// TIA Portal V19 export
FUNCTION_BLOCK "A0302_PareggiatoreCoda_FB"   // FB118, LAD
// stored: MemoryReserve 100, SetENOAutomatically false
   VAR_INPUT
      AreaInterface : "AreaInterface";
      ZSI : "udt_ZoneSafetyInterface";
      DSI_Feed : "udt_DeviceSafetyInterface";
      DSI_Valve : "udt_DeviceSafetyInterface";
      DSI_OilValve : "udt_DeviceSafetyInterface";
      Drive : "TAx_DriveInterface";
      DataIn : Struct
         OP_MoveToPos : Bool;
         BattutaVrt : Struct
            OP : "OP_PB";
         END_STRUCT;
         PareggLong : Struct
            OP : "OP_PB";
            AnalSens : Int;
         END_STRUCT;
         Sens { ExternalWritable := 'False'} : Struct
            FTC_Ingombro_In : Bool;   // 2012BF1 - I50.0
            FTC_Ingombro_Out : Bool;   // 2012BF2 - I50.1
            PresenzaMat : Bool;   // FC presenza materiale agganciato lato paregg coda
            FC_Aticoll_Spalla : Bool;
         END_STRUCT;
      END_STRUCT;
      CIn : Struct
         Manager : Struct
            EnableStopDoorOpeningReq { ExternalAccessible := 'False'; ExternalVisible := 'False'; ExternalWritable := 'False'} : Bool;
            EnableStopInPhase { ExternalAccessible := 'False'; ExternalVisible := 'False'; ExternalWritable := 'False'} : Bool;
            EnableStopProgrammed { ExternalAccessible := 'False'; ExternalVisible := 'False'; ExternalWritable := 'False'} : Bool;
            Control_ON { ExternalAccessible := 'False'; ExternalVisible := 'False'; ExternalWritable := 'False'} : Bool;
            MoveToPos { ExternalAccessible := 'False'; ExternalVisible := 'False'; ExternalWritable := 'False'} : Bool;
            Pos { ExternalAccessible := 'False'; ExternalVisible := 'False'; ExternalWritable := 'False'} : LReal;
            Speed : LReal;
            Bloccaggio { ExternalAccessible := 'False'; ExternalVisible := 'False'; ExternalWritable := 'False'} : Struct
               Rest : Bool;
               Work : Bool;
            END_STRUCT;
            BattutaVrt { ExternalAccessible := 'False'; ExternalVisible := 'False'; ExternalWritable := 'False'} : Struct
               Rest : Bool;
               Work : Bool;
            END_STRUCT;
            PareggLong { ExternalAccessible := 'False'; ExternalVisible := 'False'; ExternalWritable := 'False'} : Struct
               Rest : Bool;
               Work : Bool;
            END_STRUCT;
         END_STRUCT;
         SemiAut_Pb { ExternalWritable := 'False'} : Bool;
         Bordatrice : Struct
            Ax : "Positioning_EPOS_Machine_COut";
            Sts : Struct
               PosTargetEnable : Bool;
               PosTarget_Reached : Bool;
               In_W_Pos : Bool;
               AtRest : Bool;
            END_STRUCT;
            RegSpalla : Struct
               Infeed_ReqON : Bool;
            END_STRUCT;
         END_STRUCT;
         Rulliera { ExternalWritable := 'False'} : Struct
            Ax_1 : "SpeedMachine_COut";
            Ax_2 : "SpeedMachine_COut";
            Centratori : "ValveMachine_COut";
            Coda : Struct
               Sens : Struct
                  FTC_Rall : Bool;   // Sensori presenza materiale banco rallentamento ingresso
                  FTC_Prox_Ing : Bool;   // Sensori presenza materiale banco limite ingresso
               END_STRUCT;
            END_STRUCT;
            Centro : Struct
               Sens : Struct
                  FTC_Centrale : Bool;   // 2010BF1 - I50.2
               END_STRUCT;
            END_STRUCT;
         END_STRUCT;
         CarroPareggCoda : Struct
            Pareggia : Bool;   // Bit di abilitazione pareggiamento - prende la misura del beam e controlla la tolleranza
            OilInTargetPressure { ExternalWritable := 'False'} : Bool;
         END_STRUCT;
         CarroPareggTesta { ExternalWritable := 'False'} : Struct
            Sens : Struct
               FTC1_Rall : Bool;   // 2010BF2 - I50.3
               FTC2_Prox_Ls : Bool;   // 2010BF3 - I50.4
               PresenzaMat : Bool;   // FC presenza materiale agganciato lato paregg testa
            END_STRUCT;
         END_STRUCT;
         CarriPareggiatori : Struct
            ZoneA0302Entry_Empty { ExternalWritable := 'False'} : Bool;
            ZoneA0302Exit_Empty { ExternalWritable := 'False'} : Bool;
            RequestNewPosition : Bool;
         END_STRUCT;
         Spalle : Struct
            Coda : Struct
               ActualPos : LReal;
            END_STRUCT;
            Testa : Struct
               ActualPos : LReal;
            END_STRUCT;
         END_STRUCT;
         Manipolatore : Struct
            Sollevatore : "ValveMachine_COut";
         END_STRUCT;
         Centratori : Struct
            Sollevamento : "ValveMachine_COut";
         END_STRUCT;
      END_STRUCT;
      Config : Struct
         Ax : "Positioning_DOL_Machine_Config";
         Bloccaggio : "ValveMachine_Config";
         BattutaVerticale : "ValveMachine_Config";
         PareggiatoreLong : "ValveMachine_Config";
         PosPareggiatore : Struct
            QuotaMin_Work : LReal;
            QuotaMax_Work : LReal;
         END_STRUCT;
         MinDistanzaConSpalla : LReal;
         DelayMissingCondition : Time;
      END_STRUCT;
      HWID : Struct
         Ax_TEL1 : HW_SUBMODULE;
         Enc_IO : HW_SUBMODULE;
      END_STRUCT;
   END_VAR
   VAR_OUTPUT
      MachineInterface : "MachineInterface";
      COut : Struct
         Ax : "Positioning_DOL_Machine_COut";
         Bloccaggio : "ValveMachine_COut";
         BattutaVerticale : "ValveMachine_COut";
         PareggiatoreLong : "ValveMachine_COut";
         Ax_InWPos : Bool;
         Anticipi : Struct
            Work : Struct
               BattutaVrt : Bool;
               PareggLong : Bool;
            END_STRUCT;
            Rest : Struct
               BattutaVrt : Bool;
               PareggLong : Bool;
            END_STRUCT;
         END_STRUCT;
      END_STRUCT;
   END_VAR
   VAR_IN_OUT
      Par : Struct
         Ax : "Positioning_DOL_Machine_Par";
         Ax_Pers : "Positioning_DOL_Machine_Pers_Data";
         Enc : "PosFbk_RTN";
         Ax_Aut : "A0301_Mach_Speed_Par";
         Bloccaggio_Sens : Struct
            "2191B1" : "Analogic_SensorManagement_Par";
            SogliaWork : Real;
         END_STRUCT;
         CarroPareggCoda : Struct
            Delay_StartMove : Time;
            Preset : LReal;
         END_STRUCT;
         Cremaliera : Struct
            Modulo : LReal;
            Passo : LReal;
         END_STRUCT;
      END_STRUCT;
      Par_Sens : Struct
         AI : "Analogic_SensorManagement_Par";
      END_STRUCT;
      Data_Sens : "Analogic_SensorManagement_Data";
      Par_MachSens : "A0301_Mach_Sens_Par";
      IEC_SP : Struct
         FTC_Input : Struct
            TON_PT : Time;
            TOF_PT : Time;
         END_STRUCT;
         FTC_Output : Struct
            TON_PT : Time;
            TOF_PT : Time;
         END_STRUCT;
         FTC_PresentMat : Struct
            TON_PT : Time;
            TOF_PT : Time;
         END_STRUCT;
         Check_2119B1 : Struct
            TON_PT : Time;
         END_STRUCT;
      END_STRUCT;
   END_VAR
   VAR
      Alarm : Struct
         Ax : "Positioning_DOL_Machine_Alr";
         Enc : "PosFbk_Encoder_Alr";
         Bloccaggio : "ValveAlr";
         BattutaVerticale : "ValveAlr";
         PareggiatoreLong : "ValveAlr";
         PareggLong_AnalSens_Issue : Bool;
         SensFC_Aticoll_Spalla : Bool;
         Bloccaggio_AnalSens_Issue : Bool;   // Errore soglia lettura pressione su bloccaggio cremaliera
      END_STRUCT;
      Warning : Struct
         Ax : "Positioning_DOL_Machine_Wng";
         Bloccaggio : "ValveMachine_Wng";
         BattutaVerticale : "ValveMachine_Wng";
         PareggiatoreLongitudinale : "ValveMachine_Wng";
         PosPareggiatoreLong : "Analogic_SensorManagement_Warning";
         MissingCnd : Struct
            OP_REST_BattutaVrt : Bool;   // Mancanza comando arresto
            OP_WORK_BattutaVrt : Bool;   // Mancanza consenso lavoro
            OP_REST_PareggLong : Bool;   // Mancanza comando arresto
            OP_WORK_PareggLong : Bool;   // Mancanza consenso lavoro
            OP_REST_Bloccaggio : Bool;   // Mancanza comando arresto
            OP_WORK_Bloccaggio : Bool;   // Mancanza consenso lavoro
         END_STRUCT;
         SW_Limit_AntiCollision : Bool;
      END_STRUCT;
      HMI : Struct
         AnalogSensor : "AnalogSens_HmiData";
         Ax : Struct
            PbPreset : Bool;
            B_Preset_UM2 : Bool;
            PresetValue : LReal;
         END_STRUCT;
      END_STRUCT;
      Sts : Struct
         ReadyForMove : Bool;   // Pronto al movimento
         OP_PCoda_CanMoveFreely : Bool;
         OP_Ax_CanMoveFreely : Bool;
         Op_MoveToPos_Cnd : Bool;
         BattutaVrt : Struct
            OP_Rest_Cnd : Bool;
            Op_Work_Cnd : Bool;
         END_STRUCT;
         PareggLong : Struct
            OP_Rest_Cnd : Bool;
            Op_Work_Cnd : Bool;
         END_STRUCT;
      END_STRUCT;
      Ctrl : Struct
         BattutaVrt : Struct
            OP_Rest_Man : Bool;
            OP_Work_Man : Bool;
            OP_Rest_Aut : Bool;
            OP_Work_Aut : Bool;
            OP_Rest : Bool;
            OP_Work : Bool;
         END_STRUCT;
         PareggLong : Struct
            CheckMesure : Bool;   // Bit che determina l'uscita del pareggiatore e Controlla misura Blea nel manager
            OP_Rest_Aut : Bool;
            OP_Work_Aut : Bool;
            OP_Rest_Man : Bool;
            OP_Work_Man : Bool;
            OP_Rest : Bool;
            OP_Work : Bool;
         END_STRUCT;
         Ax : Struct
            OP_MoveToPos_Man : Bool;
            OP_MoveToPos_Aut : Bool;
            OP_MoveToPos : Bool;
         END_STRUCT;
      END_STRUCT;
      AUX : Struct
         OP_MoveToPos : Bool;
         BattutaVrt : Struct
            OP_Rest : Bool;
            OP_Work : Bool;
         END_STRUCT;
         PareggLong : Struct
            OP_Rest : Bool;
            OP_Work : Bool;
         END_STRUCT;
      END_STRUCT;
      Ax { S7_SetPoint := 'True'} : "Positioning_DOL_Machine_FB";   // Asse di movimento carro pareggiatore su cremaliera
      Enc : "PosFbk_SickAFM60";
      Enc_ITF : "PosFbk_ITF";
      Bloccaggio { S7_SetPoint := 'True'} : "ValveMachine_FB";   // Bloccaggio cremaliera
      BattutaVerticale { S7_SetPoint := 'True'} : "ValveMachine_FB";   // Battuta verticale
      PareggiatoreLong { S7_SetPoint := 'True'} : "ValveMachine_FB";   // Pareggiatore longitudinale
      PosPareggLong { S7_SetPoint := 'True'} : "Analogic_SensorManagement";   // Sensore di posizione pareggiatore
      TON_PareggLong : Struct
         OP_REST_MissingCnd { S7_SetPoint := 'True'} : TON_TIME;
         OP_WORK_MissingCnd { S7_SetPoint := 'True'} : TON_TIME;
      END_STRUCT;
      TON_BattutaVrt : Struct
         OP_REST_MissingCnd { S7_SetPoint := 'True'} : TON_TIME;
         OP_WORK_MissingCnd { S7_SetPoint := 'True'} : TON_TIME;
      END_STRUCT;
      TON_Bloccaggio : Struct
         OP_REST_MissingCnd { S7_SetPoint := 'True'} : TON_TIME;
         OP_WORK_MissingCnd { S7_SetPoint := 'True'} : TON_TIME;
      END_STRUCT;
      IEC_FTC_Input : Struct
         TON_Delay : IEC_TIMER;
         TOF_Delay { S7_SetPoint := 'True'} : IEC_TIMER;
         FTC_On { S7_SetPoint := 'True'} : Bool;
      END_STRUCT;
      IEC_FTC_Output : Struct
         TON_Delay : IEC_TIMER;
         TOF_Delay { S7_SetPoint := 'True'} : IEC_TIMER;
         FTC_On { S7_SetPoint := 'True'} : Bool;
      END_STRUCT;
      IEC_FTC_PresentMat : Struct
         TON_Delay : IEC_TIMER;
         TOF_Delay { S7_SetPoint := 'True'} : IEC_TIMER;
         FTC_On { S7_SetPoint := 'True'} : Bool;
      END_STRUCT;
      IEC_DelayCheck_2119B1 : IEC_TIMER;
      Bloccaggio_AnalSens { S7_SetPoint := 'True'} : "AnalogThreshold";
      CarroCoda { ExternalAccessible := 'False'; ExternalVisible := 'False'; ExternalWritable := 'False'} : Struct
         RimanenzaPos : LReal;
         PassoReq : LReal;
         PosBattutePz : LReal;
         SemiBeamLen : LReal;
         NrPassiReq : LReal;
         Pos : LReal;   // Posizione calcolata in funzione della cremaliera
      END_STRUCT;
      TON_DistanzaOK : IEC_TIMER;
      TON_Anticipi : Struct
         Rest : Struct
            BattutaVrt { S7_SetPoint := 'True'} : IEC_TIMER;
            PareggLong : IEC_TIMER;
         END_STRUCT;
         Work : Struct
            PareggLong : IEC_TIMER;
            BattutaVrt { S7_SetPoint := 'True'} : IEC_TIMER;
         END_STRUCT;
      END_STRUCT;
   END_VAR
   VAR_TEMP
      PE : Struct
         OP_MoveToPos : Bool;
         BattutaVrt : Struct
            OP_Rest : Bool;
            OP_Work : Bool;
         END_STRUCT;
         PareggLong : Struct
            OP_Rest : Bool;
            OP_Work : Bool;
         END_STRUCT;
      END_STRUCT;
      ActualDifference : LReal;
   END_VAR
   VAR CONSTANT
      RACK_STEP : LReal;   // Passo Cremagliera mm
   END_VAR
   VAR_TEMP   // added for the SCL form of the ladder/FBD networks
      _w1 : Bool;
      _w2 : Bool;
      _w3 : Bool;
      _w4 : Bool;
      _w5 : Bool;
      _w6 : Bool;
      _w7 : Bool;
      _w8 : Bool;
      _w9 : Bool;
      _w10 : Bool;
      _w11 : Bool;
      _w12 : Bool;
   END_VAR
BEGIN

REGION Network 1 (SCL): Reset allarmi
   IF #AreaInterface.RstAlarms THEN
       #Alarm.PareggLong_AnalSens_Issue := FALSE;
       #Alarm.SensFC_Aticoll_Spalla := FALSE;
       #Alarm.Bloccaggio_AnalSens_Issue := FALSE;
   END_IF;
END_REGION

REGION Network 2: <+>
END_REGION

REGION Network 3: Anticipi Movimento LAVORO
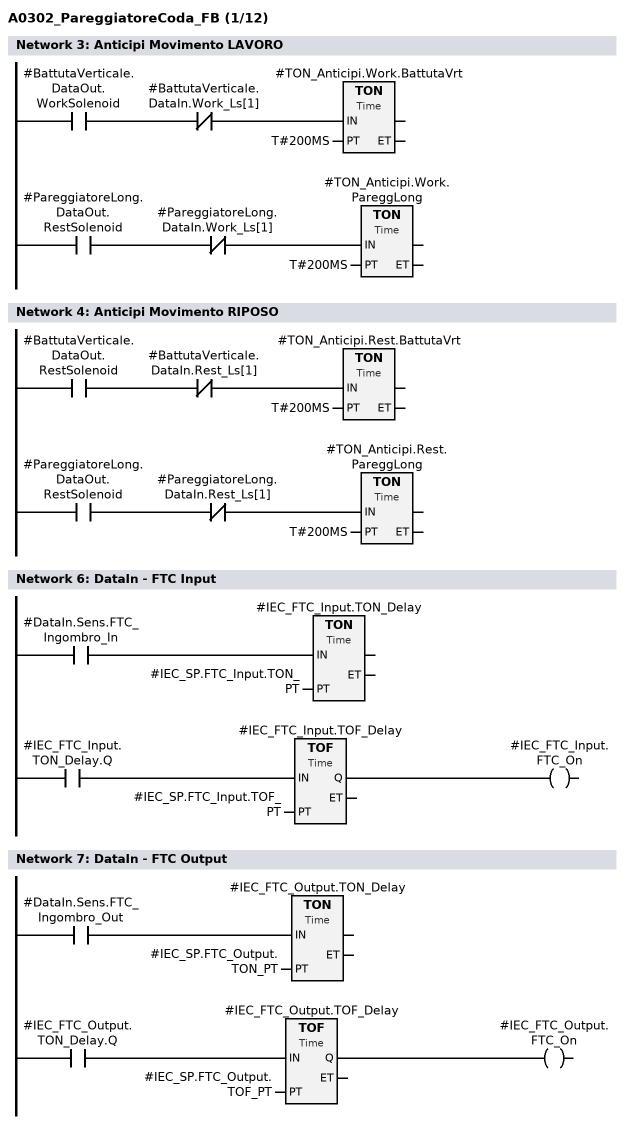
   RUNG wire#powerrail
      Contact( #BattutaVerticale.DataOut.WorkSolenoid )
      I_Contact( #BattutaVerticale.DataIn.Work_Ls[1] )
      { S7_Templates := "time_type := Time" } #TON_Anticipi.Work.BattutaVrt.TON(pt := T#200MS, et =>)
   END_RUNG
   RUNG wire#powerrail
      Contact( #PareggiatoreLong.DataOut.RestSolenoid )
      I_Contact( #PareggiatoreLong.DataIn.Work_Ls[1] )
      { S7_Templates := "time_type := Time" } #TON_Anticipi.Work.PareggLong.TON(pt := T#200MS, et =>)
   END_RUNG
   // the same network as SCL:
   #TON_Anticipi.Work.BattutaVrt.TON(IN := #BattutaVerticale.DataOut.WorkSolenoid AND NOT #BattutaVerticale.DataIn.Work_Ls[1],
                           PT := T#200MS);
   #TON_Anticipi.Work.PareggLong.TON(IN := #PareggiatoreLong.DataOut.RestSolenoid AND NOT #PareggiatoreLong.DataIn.Work_Ls[1],
                           PT := T#200MS);
END_REGION

REGION Network 4: Anticipi Movimento RIPOSO
   RUNG wire#powerrail
      Contact( #BattutaVerticale.DataOut.RestSolenoid )
      I_Contact( #BattutaVerticale.DataIn.Rest_Ls[1] )
      { S7_Templates := "time_type := Time" } #TON_Anticipi.Rest.BattutaVrt.TON(pt := T#200MS, et =>)
   END_RUNG
   RUNG wire#powerrail
      Contact( #PareggiatoreLong.DataOut.RestSolenoid )
      I_Contact( #PareggiatoreLong.DataIn.Rest_Ls[1] )
      { S7_Templates := "time_type := Time" } #TON_Anticipi.Rest.PareggLong.TON(pt := T#200MS, et =>)
   END_RUNG
   // the same network as SCL:
   #TON_Anticipi.Rest.BattutaVrt.TON(IN := #BattutaVerticale.DataOut.RestSolenoid AND NOT #BattutaVerticale.DataIn.Rest_Ls[1],
                           PT := T#200MS);
   #TON_Anticipi.Rest.PareggLong.TON(IN := #PareggiatoreLong.DataOut.RestSolenoid AND NOT #PareggiatoreLong.DataIn.Rest_Ls[1],
                           PT := T#200MS);
END_REGION

REGION Network 5: <+>
END_REGION

REGION Network 6: DataIn - FTC Input
   RUNG wire#powerrail
      Contact( #DataIn.Sens.FTC_Ingombro_In )
      { S7_Templates := "time_type := Time" } #IEC_FTC_Input.TON_Delay.TON(pt := #IEC_SP.FTC_Input.TON_PT, et =>)
   END_RUNG
   RUNG wire#powerrail
      Contact( #IEC_FTC_Input.TON_Delay.Q )
      { S7_Templates := "time_type := Time" } #IEC_FTC_Input.TOF_Delay.TOF(pt := #IEC_SP.FTC_Input.TOF_PT, et =>)
      Coil( #IEC_FTC_Input.FTC_On )
   END_RUNG
   // the same network as SCL:
   #IEC_FTC_Input.TON_Delay.TON(IN := #DataIn.Sens.FTC_Ingombro_In, PT := #IEC_SP.FTC_Input.TON_PT);
   #IEC_FTC_Input.TOF_Delay.TOF(IN := #IEC_FTC_Input.TON_Delay.Q, PT := #IEC_SP.FTC_Input.TOF_PT);
   #IEC_FTC_Input.FTC_On := #IEC_FTC_Input.TOF_Delay.Q;
END_REGION

REGION Network 7: DataIn - FTC Output
   RUNG wire#powerrail
      Contact( #DataIn.Sens.FTC_Ingombro_Out )
      { S7_Templates := "time_type := Time" } #IEC_FTC_Output.TON_Delay.TON(pt := #IEC_SP.FTC_Output.TON_PT, et =>)
   END_RUNG
   RUNG wire#powerrail
      Contact( #IEC_FTC_Output.TON_Delay.Q )
      { S7_Templates := "time_type := Time" } #IEC_FTC_Output.TOF_Delay.TOF(pt := #IEC_SP.FTC_Output.TOF_PT, et =>)
      Coil( #IEC_FTC_Output.FTC_On )
   END_RUNG
   // the same network as SCL:
   #IEC_FTC_Output.TON_Delay.TON(IN := #DataIn.Sens.FTC_Ingombro_Out, PT := #IEC_SP.FTC_Output.TON_PT);
   #IEC_FTC_Output.TOF_Delay.TOF(IN := #IEC_FTC_Output.TON_Delay.Q, PT := #IEC_SP.FTC_Output.TOF_PT);
   #IEC_FTC_Output.FTC_On := #IEC_FTC_Output.TOF_Delay.Q;
END_REGION

REGION Network 8: DataIn - FTC Presenza materiale
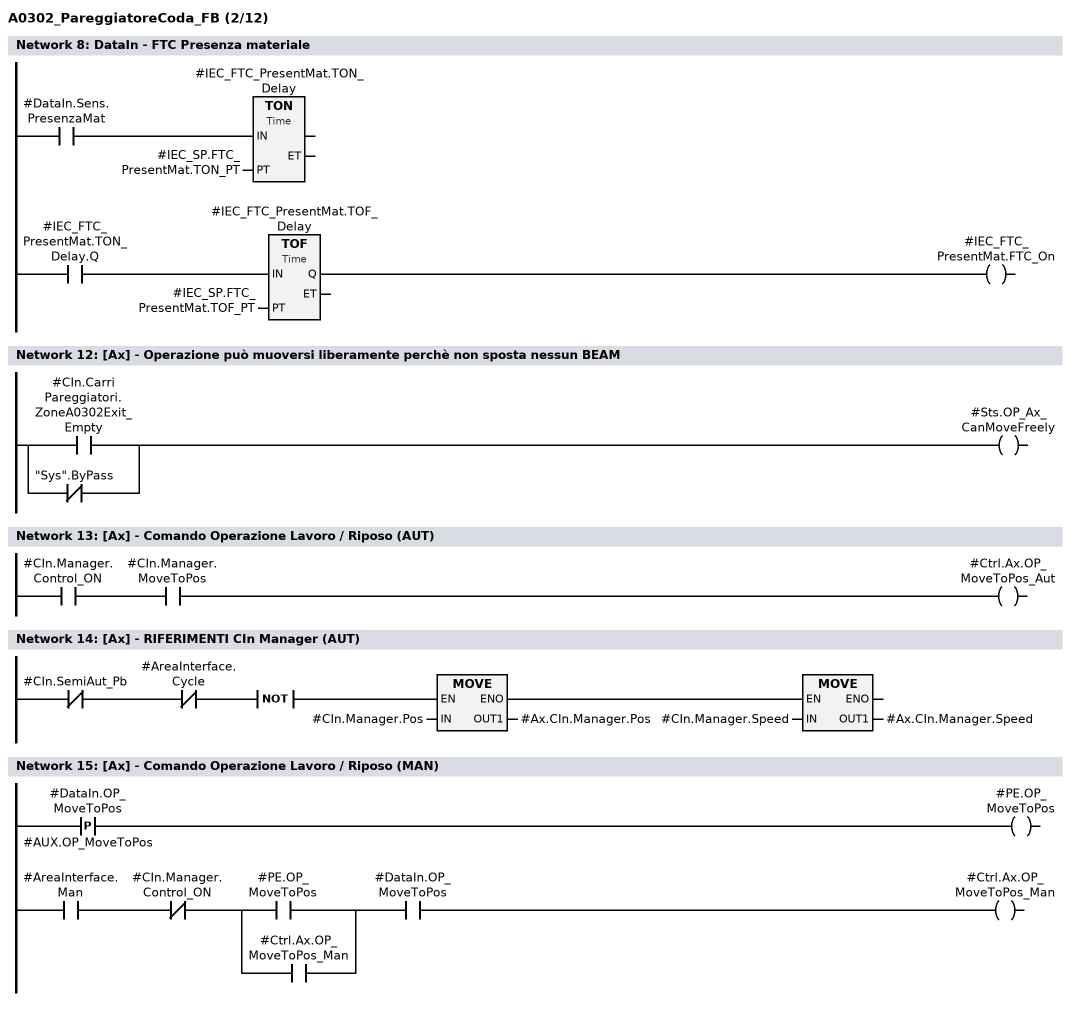
   RUNG wire#powerrail
      Contact( #DataIn.Sens.PresenzaMat )
      { S7_Templates := "time_type := Time" } #IEC_FTC_PresentMat.TON_Delay.TON(pt := #IEC_SP.FTC_PresentMat.TON_PT, et =>)
   END_RUNG
   RUNG wire#powerrail
      Contact( #IEC_FTC_PresentMat.TON_Delay.Q )
      { S7_Templates := "time_type := Time" } #IEC_FTC_PresentMat.TOF_Delay.TOF(pt := #IEC_SP.FTC_PresentMat.TOF_PT, et =>)
      Coil( #IEC_FTC_PresentMat.FTC_On )
   END_RUNG
   // the same network as SCL:
   #IEC_FTC_PresentMat.TON_Delay.TON(IN := #DataIn.Sens.PresenzaMat, PT := #IEC_SP.FTC_PresentMat.TON_PT);
   #IEC_FTC_PresentMat.TOF_Delay.TOF(IN := #IEC_FTC_PresentMat.TON_Delay.Q, PT := #IEC_SP.FTC_PresentMat.TOF_PT);
   #IEC_FTC_PresentMat.FTC_On := #IEC_FTC_PresentMat.TOF_Delay.Q;
END_REGION

REGION Network 9: <+>
END_REGION

REGION Network 10: <<< CARRO PAREGGIATORE CODA >>>
END_REGION

REGION Network 11: <+>
END_REGION

REGION Network 12: [Ax] - Operazione può muoversi liberamente perchè non sposta nessun BEAM
   RUNG wire#powerrail
      Contact( #CIn.CarriPareggiatori.ZoneA0302Exit_Empty )
      wire#w1
      Coil( #Sts.OP_Ax_CanMoveFreely )
   END_RUNG
   RUNG wire#powerrail
      I_Contact( "Sys".ByPass )
   END_RUNG wire#w1
   // the same network as SCL:
   #Sts.OP_Ax_CanMoveFreely := #CIn.CarriPareggiatori.ZoneA0302Exit_Empty OR NOT "Sys".ByPass;
END_REGION

REGION Network 13: [Ax] - Comando Operazione Lavoro / Riposo (AUT)
   RUNG wire#powerrail
      Contact( #CIn.Manager.Control_ON )
      Contact( #CIn.Manager.MoveToPos )
      Coil( #Ctrl.Ax.OP_MoveToPos_Aut )
   END_RUNG
   // the same network as SCL:
   #Ctrl.Ax.OP_MoveToPos_Aut := #CIn.Manager.Control_ON AND #CIn.Manager.MoveToPos;
END_REGION

REGION Network 14: [Ax] - RIFERIMENTI CIn Manager (AUT)
   RUNG wire#powerrail
      I_Contact( #CIn.SemiAut_Pb )
      I_Contact( #AreaInterface.Cycle )
      Not()
      Move(in := #CIn.Manager.Pos, out1 => #Ax.CIn.Manager.Pos)
      Move(in := #CIn.Manager.Speed, out1 => #Ax.CIn.Manager.Speed)
   END_RUNG
   // the same network as SCL:
   IF NOT (NOT #CIn.SemiAut_Pb AND NOT #AreaInterface.Cycle) THEN
       #Ax.CIn.Manager.Pos := #CIn.Manager.Pos;
       #Ax.CIn.Manager.Speed := #CIn.Manager.Speed;
   END_IF;
END_REGION

REGION Network 15: [Ax] - Comando Operazione Lavoro / Riposo (MAN)
   RUNG wire#powerrail
      P_Contact(operand := #DataIn.OP_MoveToPos, bit := #AUX.OP_MoveToPos)
      Coil( #PE.OP_MoveToPos )
   END_RUNG
   RUNG wire#powerrail
      Contact( #AreaInterface.Man )
      I_Contact( #CIn.Manager.Control_ON )
      wire#w1
      Contact( #PE.OP_MoveToPos )
      wire#w2
      Contact( #DataIn.OP_MoveToPos )
      Coil( #Ctrl.Ax.OP_MoveToPos_Man )
   END_RUNG
   RUNG wire#w1
      Contact( #Ctrl.Ax.OP_MoveToPos_Man )
   END_RUNG wire#w2
   // the same network as SCL:
   #_w1 := #DataIn.OP_MoveToPos AND NOT #AUX.OP_MoveToPos;   // rising edge of #DataIn.OP_MoveToPos
   #AUX.OP_MoveToPos := #DataIn.OP_MoveToPos;
   #PE.OP_MoveToPos := #_w1;
   #Ctrl.Ax.OP_MoveToPos_Man := #AreaInterface.Man AND NOT #CIn.Manager.Control_ON AND (#PE.OP_MoveToPos OR #Ctrl.Ax.OP_MoveToPos_Man) AND #DataIn.OP_MoveToPos;
END_REGION

REGION Network 16: <+>
END_REGION

REGION Network 17: [Battuta Vrt + Paregg. Long] - Operazione può muoversi liberamente perchè non sposta nessun BEAM
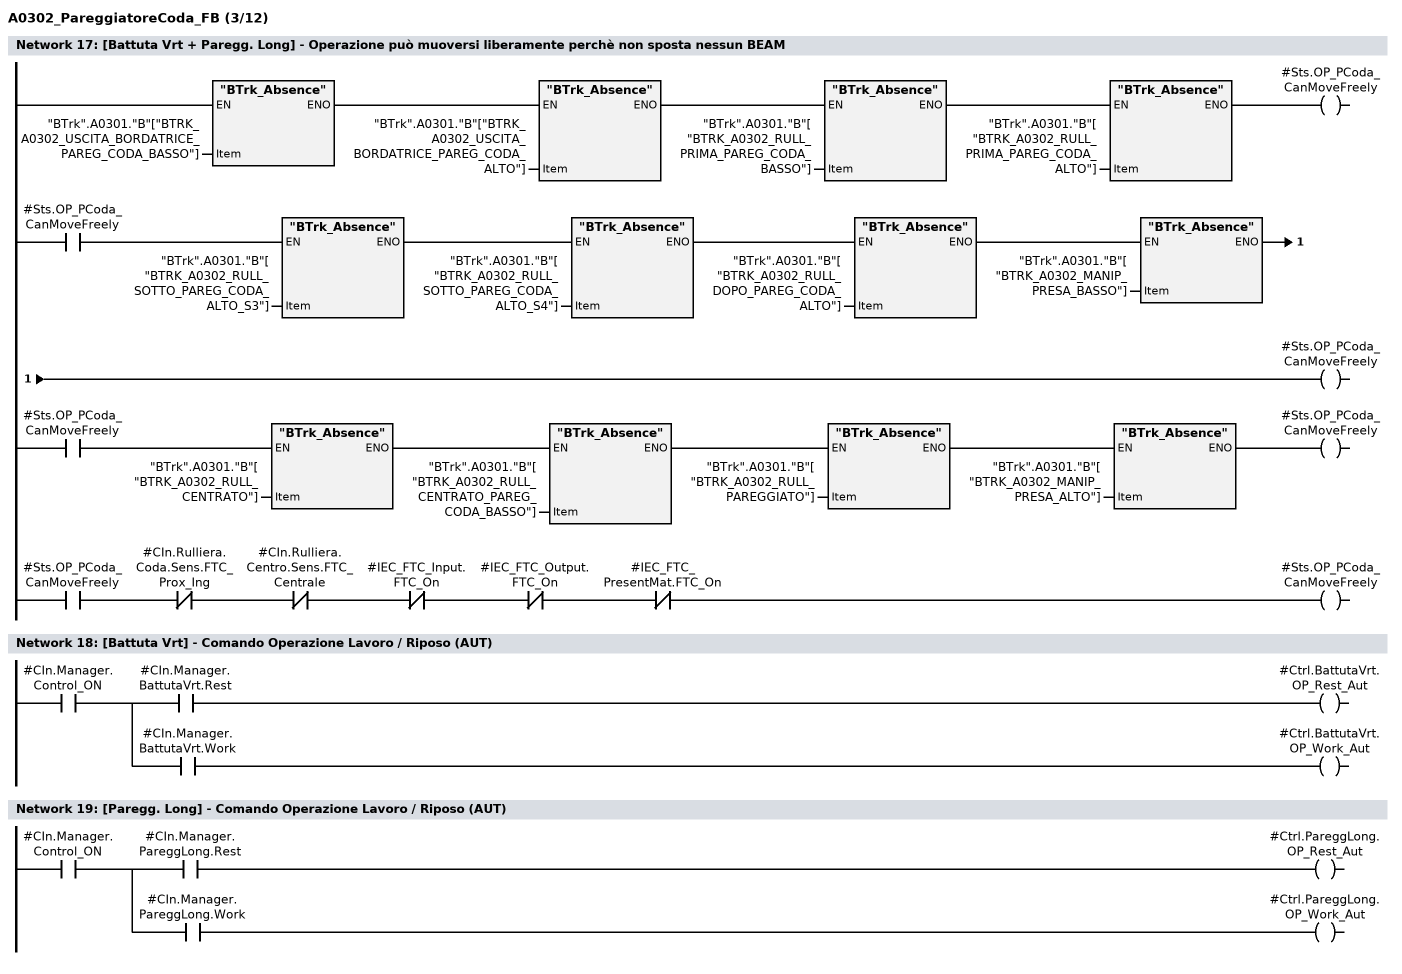
   RUNG wire#powerrail
      "BTrk_Absence"(Item := "BTrk".A0301."B"["BTRK_A0302_USCITA_BORDATRICE_PAREG_CODA_BASSO"])
      "BTrk_Absence"(Item := "BTrk".A0301."B"["BTRK_A0302_USCITA_BORDATRICE_PAREG_CODA_ALTO"])
      "BTrk_Absence"(Item := "BTrk".A0301."B"["BTRK_A0302_RULL_PRIMA_PAREG_CODA_BASSO"])
      "BTrk_Absence"(Item := "BTrk".A0301."B"["BTRK_A0302_RULL_PRIMA_PAREG_CODA_ALTO"])
      Coil( #Sts.OP_PCoda_CanMoveFreely )
   END_RUNG
   RUNG wire#powerrail
      Contact( #Sts.OP_PCoda_CanMoveFreely )
      "BTrk_Absence"(Item := "BTrk".A0301."B"["BTRK_A0302_RULL_SOTTO_PAREG_CODA_ALTO_S3"])
      "BTrk_Absence"(Item := "BTrk".A0301."B"["BTRK_A0302_RULL_SOTTO_PAREG_CODA_ALTO_S4"])
      "BTrk_Absence"(Item := "BTrk".A0301."B"["BTRK_A0302_RULL_DOPO_PAREG_CODA_ALTO"])
      "BTrk_Absence"(Item := "BTrk".A0301."B"["BTRK_A0302_MANIP_PRESA_BASSO"])
      Coil( #Sts.OP_PCoda_CanMoveFreely )
   END_RUNG
   RUNG wire#powerrail
      Contact( #Sts.OP_PCoda_CanMoveFreely )
      "BTrk_Absence"(Item := "BTrk".A0301."B"["BTRK_A0302_RULL_CENTRATO"])
      "BTrk_Absence"(Item := "BTrk".A0301."B"["BTRK_A0302_RULL_CENTRATO_PAREG_CODA_BASSO"])
      "BTrk_Absence"(Item := "BTrk".A0301."B"["BTRK_A0302_RULL_PAREGGIATO"])
      "BTrk_Absence"(Item := "BTrk".A0301."B"["BTRK_A0302_MANIP_PRESA_ALTO"])
      Coil( #Sts.OP_PCoda_CanMoveFreely )
   END_RUNG
   RUNG wire#powerrail
      Contact( #Sts.OP_PCoda_CanMoveFreely )
      I_Contact( #CIn.Rulliera.Coda.Sens.FTC_Prox_Ing )
      I_Contact( #CIn.Rulliera.Centro.Sens.FTC_Centrale )
      I_Contact( #IEC_FTC_Input.FTC_On )
      I_Contact( #IEC_FTC_Output.FTC_On )
      I_Contact( #IEC_FTC_PresentMat.FTC_On )
      Coil( #Sts.OP_PCoda_CanMoveFreely )
   END_RUNG
   // the same network as SCL:
   "BTrk_Absence"(Item := "BTrk".A0301."B"["BTRK_A0302_USCITA_BORDATRICE_PAREG_CODA_BASSO"], ENO => #_w1);
   "BTrk_Absence"(EN := #_w1,
                  Item := "BTrk".A0301."B"["BTRK_A0302_USCITA_BORDATRICE_PAREG_CODA_ALTO"],
                  ENO => #_w2);
   "BTrk_Absence"(EN := #_w2, Item := "BTrk".A0301."B"["BTRK_A0302_RULL_PRIMA_PAREG_CODA_BASSO"], ENO => #_w3);
   "BTrk_Absence"(EN := #_w3, Item := "BTrk".A0301."B"["BTRK_A0302_RULL_PRIMA_PAREG_CODA_ALTO"], ENO => #_w4);
   #Sts.OP_PCoda_CanMoveFreely := #_w4;
   "BTrk_Absence"(EN := #Sts.OP_PCoda_CanMoveFreely,
                  Item := "BTrk".A0301."B"["BTRK_A0302_RULL_SOTTO_PAREG_CODA_ALTO_S3"],
                  ENO => #_w5);
   "BTrk_Absence"(EN := #_w5, Item := "BTrk".A0301."B"["BTRK_A0302_RULL_SOTTO_PAREG_CODA_ALTO_S4"], ENO => #_w6);
   "BTrk_Absence"(EN := #_w6, Item := "BTrk".A0301."B"["BTRK_A0302_RULL_DOPO_PAREG_CODA_ALTO"], ENO => #_w7);
   "BTrk_Absence"(EN := #_w7, Item := "BTrk".A0301."B"["BTRK_A0302_MANIP_PRESA_BASSO"], ENO => #_w8);
   #Sts.OP_PCoda_CanMoveFreely := #_w8;
   "BTrk_Absence"(EN := #Sts.OP_PCoda_CanMoveFreely,
                  Item := "BTrk".A0301."B"["BTRK_A0302_RULL_CENTRATO"],
                  ENO => #_w9);
   "BTrk_Absence"(EN := #_w9,
                  Item := "BTrk".A0301."B"["BTRK_A0302_RULL_CENTRATO_PAREG_CODA_BASSO"],
                  ENO => #_w10);
   "BTrk_Absence"(EN := #_w10, Item := "BTrk".A0301."B"["BTRK_A0302_RULL_PAREGGIATO"], ENO => #_w11);
   "BTrk_Absence"(EN := #_w11, Item := "BTrk".A0301."B"["BTRK_A0302_MANIP_PRESA_ALTO"], ENO => #_w12);
   #Sts.OP_PCoda_CanMoveFreely := #_w12;
   #Sts.OP_PCoda_CanMoveFreely := #Sts.OP_PCoda_CanMoveFreely AND NOT #CIn.Rulliera.Coda.Sens.FTC_Prox_Ing AND NOT #CIn.Rulliera.Centro.Sens.FTC_Centrale AND NOT #IEC_FTC_Input.FTC_On AND NOT #IEC_FTC_Output.FTC_On AND NOT #IEC_FTC_PresentMat.FTC_On;
END_REGION

REGION Network 18: [Battuta Vrt] - Comando Operazione Lavoro / Riposo (AUT)
   RUNG wire#powerrail
      Contact( #CIn.Manager.Control_ON )
      wire#w1
      Contact( #CIn.Manager.BattutaVrt.Rest )
      Coil( #Ctrl.BattutaVrt.OP_Rest_Aut )
   END_RUNG
   RUNG wire#w1
      Contact( #CIn.Manager.BattutaVrt.Work )
      Coil( #Ctrl.BattutaVrt.OP_Work_Aut )
   END_RUNG
   // the same network as SCL:
   #Ctrl.BattutaVrt.OP_Rest_Aut := #CIn.Manager.Control_ON AND #CIn.Manager.BattutaVrt.Rest;
   #Ctrl.BattutaVrt.OP_Work_Aut := #CIn.Manager.Control_ON AND #CIn.Manager.BattutaVrt.Work;
END_REGION

REGION Network 19: [Paregg. Long] - Comando Operazione Lavoro / Riposo (AUT)
   RUNG wire#powerrail
      Contact( #CIn.Manager.Control_ON )
      wire#w1
      Contact( #CIn.Manager.PareggLong.Rest )
      Coil( #Ctrl.PareggLong.OP_Rest_Aut )
   END_RUNG
   RUNG wire#w1
      Contact( #CIn.Manager.PareggLong.Work )
      Coil( #Ctrl.PareggLong.OP_Work_Aut )
   END_RUNG
   // the same network as SCL:
   #Ctrl.PareggLong.OP_Rest_Aut := #CIn.Manager.Control_ON AND #CIn.Manager.PareggLong.Rest;
   #Ctrl.PareggLong.OP_Work_Aut := #CIn.Manager.Control_ON AND #CIn.Manager.PareggLong.Work;
END_REGION

REGION Network 20: <+>
END_REGION

REGION Network 21: [Battuta Vrt] - Comando Operazione Lavoro / Riposo (MAN)
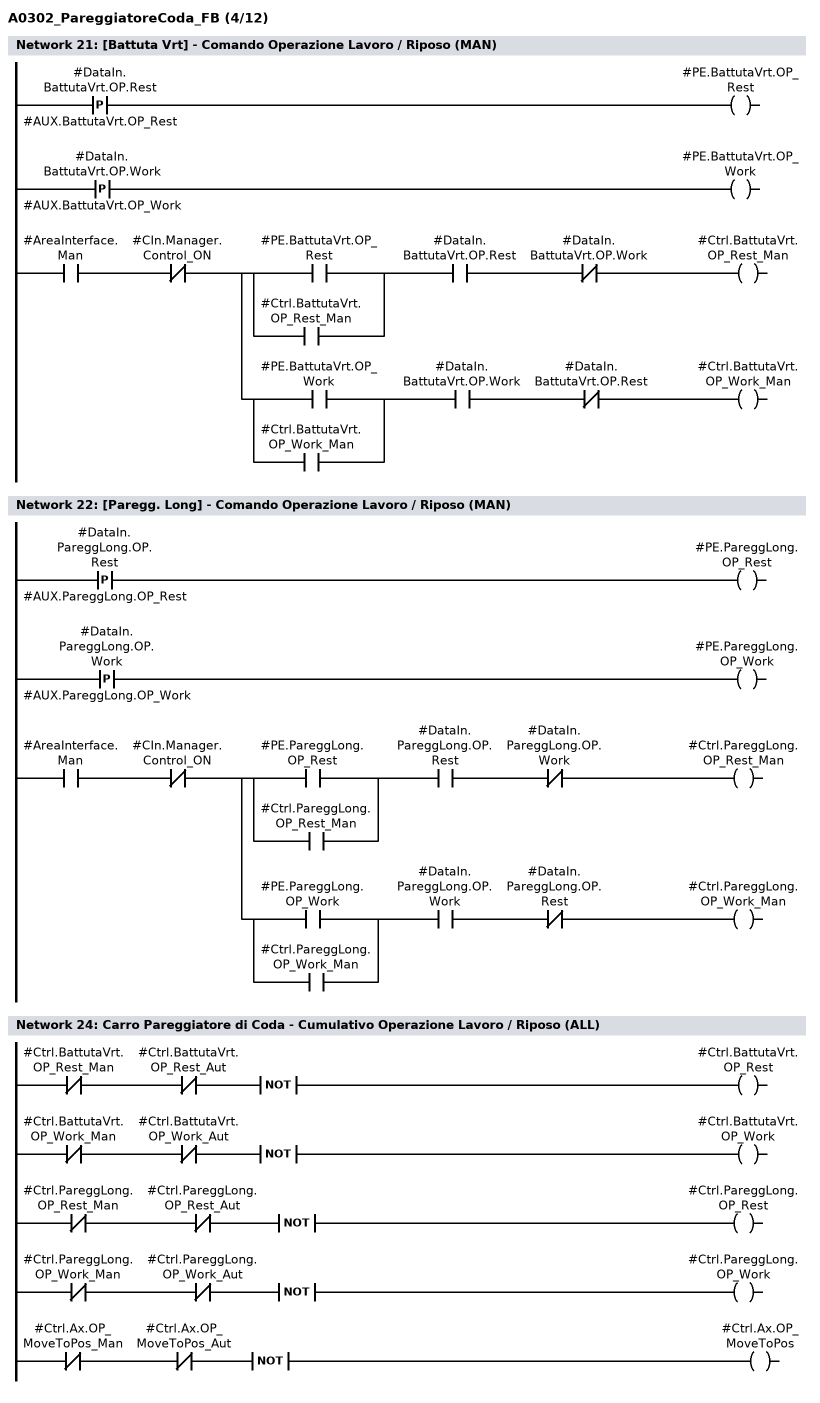
   RUNG wire#powerrail
      P_Contact(operand := #DataIn.BattutaVrt.OP.Rest, bit := #AUX.BattutaVrt.OP_Rest)
      Coil( #PE.BattutaVrt.OP_Rest )
   END_RUNG
   RUNG wire#powerrail
      P_Contact(operand := #DataIn.BattutaVrt.OP.Work, bit := #AUX.BattutaVrt.OP_Work)
      Coil( #PE.BattutaVrt.OP_Work )
   END_RUNG
   RUNG wire#powerrail
      Contact( #AreaInterface.Man )
      I_Contact( #CIn.Manager.Control_ON )
      wire#w1
      Contact( #PE.BattutaVrt.OP_Rest )
      wire#w2
      Contact( #DataIn.BattutaVrt.OP.Rest )
      I_Contact( #DataIn.BattutaVrt.OP.Work )
      Coil( #Ctrl.BattutaVrt.OP_Rest_Man )
   END_RUNG
   RUNG wire#w1
      Contact( #Ctrl.BattutaVrt.OP_Rest_Man )
   END_RUNG wire#w2
   RUNG wire#w1
      Contact( #PE.BattutaVrt.OP_Work )
      wire#w3
      Contact( #DataIn.BattutaVrt.OP.Work )
      I_Contact( #DataIn.BattutaVrt.OP.Rest )
      Coil( #Ctrl.BattutaVrt.OP_Work_Man )
   END_RUNG
   RUNG wire#w1
      Contact( #Ctrl.BattutaVrt.OP_Work_Man )
   END_RUNG wire#w3
   // the same network as SCL:
   #_w1 := #DataIn.BattutaVrt.OP.Rest AND NOT #AUX.BattutaVrt.OP_Rest;   // rising edge of #DataIn.BattutaVrt.OP.Rest
   #AUX.BattutaVrt.OP_Rest := #DataIn.BattutaVrt.OP.Rest;
   #PE.BattutaVrt.OP_Rest := #_w1;
   #_w2 := #DataIn.BattutaVrt.OP.Work AND NOT #AUX.BattutaVrt.OP_Work;   // rising edge of #DataIn.BattutaVrt.OP.Work
   #AUX.BattutaVrt.OP_Work := #DataIn.BattutaVrt.OP.Work;
   #PE.BattutaVrt.OP_Work := #_w2;
   #_w3 := #AreaInterface.Man AND NOT #CIn.Manager.Control_ON;
   #Ctrl.BattutaVrt.OP_Rest_Man := #_w3 AND (#PE.BattutaVrt.OP_Rest OR #Ctrl.BattutaVrt.OP_Rest_Man) AND #DataIn.BattutaVrt.OP.Rest AND NOT #DataIn.BattutaVrt.OP.Work;
   #Ctrl.BattutaVrt.OP_Work_Man := #_w3 AND (#PE.BattutaVrt.OP_Work OR #Ctrl.BattutaVrt.OP_Work_Man) AND #DataIn.BattutaVrt.OP.Work AND NOT #DataIn.BattutaVrt.OP.Rest;
END_REGION

REGION Network 22: [Paregg. Long] - Comando Operazione Lavoro / Riposo (MAN)
   RUNG wire#powerrail
      P_Contact(operand := #DataIn.PareggLong.OP.Rest, bit := #AUX.PareggLong.OP_Rest)
      Coil( #PE.PareggLong.OP_Rest )
   END_RUNG
   RUNG wire#powerrail
      P_Contact(operand := #DataIn.PareggLong.OP.Work, bit := #AUX.PareggLong.OP_Work)
      Coil( #PE.PareggLong.OP_Work )
   END_RUNG
   RUNG wire#powerrail
      Contact( #AreaInterface.Man )
      I_Contact( #CIn.Manager.Control_ON )
      wire#w1
      Contact( #PE.PareggLong.OP_Rest )
      wire#w2
      Contact( #DataIn.PareggLong.OP.Rest )
      I_Contact( #DataIn.PareggLong.OP.Work )
      Coil( #Ctrl.PareggLong.OP_Rest_Man )
   END_RUNG
   RUNG wire#w1
      Contact( #Ctrl.PareggLong.OP_Rest_Man )
   END_RUNG wire#w2
   RUNG wire#w1
      Contact( #PE.PareggLong.OP_Work )
      wire#w3
      Contact( #DataIn.PareggLong.OP.Work )
      I_Contact( #DataIn.PareggLong.OP.Rest )
      Coil( #Ctrl.PareggLong.OP_Work_Man )
   END_RUNG
   RUNG wire#w1
      Contact( #Ctrl.PareggLong.OP_Work_Man )
   END_RUNG wire#w3
   // the same network as SCL:
   #_w1 := #DataIn.PareggLong.OP.Rest AND NOT #AUX.PareggLong.OP_Rest;   // rising edge of #DataIn.PareggLong.OP.Rest
   #AUX.PareggLong.OP_Rest := #DataIn.PareggLong.OP.Rest;
   #PE.PareggLong.OP_Rest := #_w1;
   #_w2 := #DataIn.PareggLong.OP.Work AND NOT #AUX.PareggLong.OP_Work;   // rising edge of #DataIn.PareggLong.OP.Work
   #AUX.PareggLong.OP_Work := #DataIn.PareggLong.OP.Work;
   #PE.PareggLong.OP_Work := #_w2;
   #_w3 := #AreaInterface.Man AND NOT #CIn.Manager.Control_ON;
   #Ctrl.PareggLong.OP_Rest_Man := #_w3 AND (#PE.PareggLong.OP_Rest OR #Ctrl.PareggLong.OP_Rest_Man) AND #DataIn.PareggLong.OP.Rest AND NOT #DataIn.PareggLong.OP.Work;
   #Ctrl.PareggLong.OP_Work_Man := #_w3 AND (#PE.PareggLong.OP_Work OR #Ctrl.PareggLong.OP_Work_Man) AND #DataIn.PareggLong.OP.Work AND NOT #DataIn.PareggLong.OP.Rest;
END_REGION

REGION Network 23: <+>
END_REGION

REGION Network 24: Carro Pareggiatore di Coda - Cumulativo Operazione Lavoro / Riposo (ALL)
   RUNG wire#powerrail
      I_Contact( #Ctrl.BattutaVrt.OP_Rest_Man )
      I_Contact( #Ctrl.BattutaVrt.OP_Rest_Aut )
      Not()
      Coil( #Ctrl.BattutaVrt.OP_Rest )
   END_RUNG
   RUNG wire#powerrail
      I_Contact( #Ctrl.BattutaVrt.OP_Work_Man )
      I_Contact( #Ctrl.BattutaVrt.OP_Work_Aut )
      Not()
      Coil( #Ctrl.BattutaVrt.OP_Work )
   END_RUNG
   RUNG wire#powerrail
      I_Contact( #Ctrl.PareggLong.OP_Rest_Man )
      I_Contact( #Ctrl.PareggLong.OP_Rest_Aut )
      Not()
      Coil( #Ctrl.PareggLong.OP_Rest )
   END_RUNG
   RUNG wire#powerrail
      I_Contact( #Ctrl.PareggLong.OP_Work_Man )
      I_Contact( #Ctrl.PareggLong.OP_Work_Aut )
      Not()
      Coil( #Ctrl.PareggLong.OP_Work )
   END_RUNG
   RUNG wire#powerrail
      I_Contact( #Ctrl.Ax.OP_MoveToPos_Man )
      I_Contact( #Ctrl.Ax.OP_MoveToPos_Aut )
      Not()
      Coil( #Ctrl.Ax.OP_MoveToPos )
   END_RUNG
   // the same network as SCL:
   #Ctrl.BattutaVrt.OP_Rest := NOT (NOT #Ctrl.BattutaVrt.OP_Rest_Man AND NOT #Ctrl.BattutaVrt.OP_Rest_Aut);
   #Ctrl.BattutaVrt.OP_Work := NOT (NOT #Ctrl.BattutaVrt.OP_Work_Man AND NOT #Ctrl.BattutaVrt.OP_Work_Aut);
   #Ctrl.PareggLong.OP_Rest := NOT (NOT #Ctrl.PareggLong.OP_Rest_Man AND NOT #Ctrl.PareggLong.OP_Rest_Aut);
   #Ctrl.PareggLong.OP_Work := NOT (NOT #Ctrl.PareggLong.OP_Work_Man AND NOT #Ctrl.PareggLong.OP_Work_Aut);
   #Ctrl.Ax.OP_MoveToPos := NOT (NOT #Ctrl.Ax.OP_MoveToPos_Man AND NOT #Ctrl.Ax.OP_MoveToPos_Aut);
END_REGION

REGION Network 25: <+>
END_REGION

REGION Network 26: [Ax] - Condizioni movimento Operazione a Lavoro / Riposo
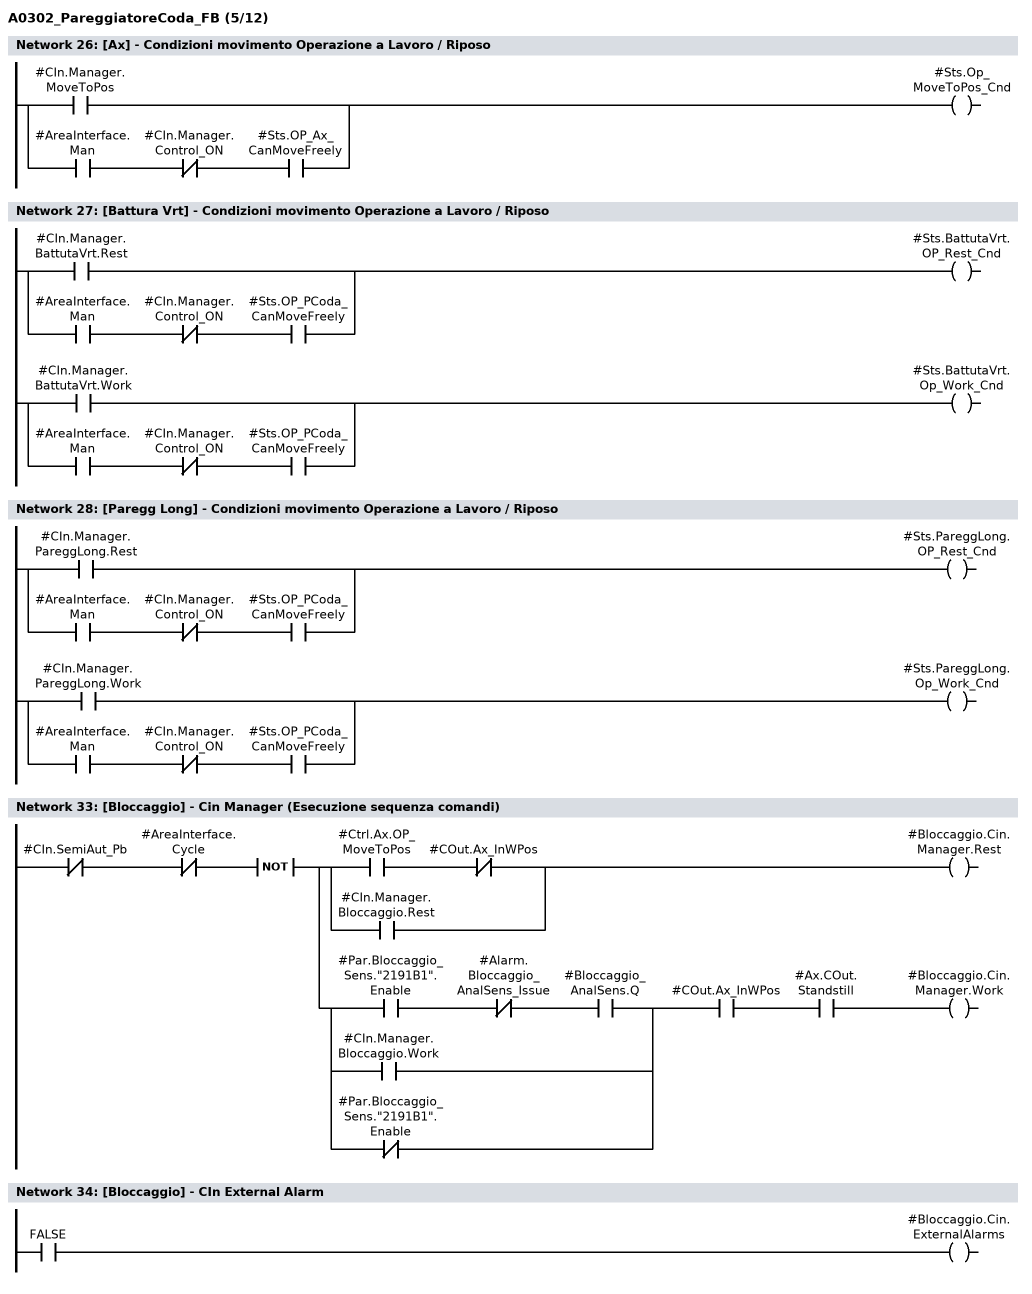
   RUNG wire#powerrail
      Contact( #CIn.Manager.MoveToPos )
      wire#w1
      Coil( #Sts.Op_MoveToPos_Cnd )
   END_RUNG
   RUNG wire#powerrail
      Contact( #AreaInterface.Man )
      I_Contact( #CIn.Manager.Control_ON )
      Contact( #Sts.OP_Ax_CanMoveFreely )
   END_RUNG wire#w1
   // the same network as SCL:
   #Sts.Op_MoveToPos_Cnd := #CIn.Manager.MoveToPos OR (#AreaInterface.Man AND NOT #CIn.Manager.Control_ON AND #Sts.OP_Ax_CanMoveFreely);
END_REGION

REGION Network 27: [Battura Vrt] - Condizioni movimento Operazione a Lavoro / Riposo
   RUNG wire#powerrail
      Contact( #CIn.Manager.BattutaVrt.Rest )
      wire#w1
      Coil( #Sts.BattutaVrt.OP_Rest_Cnd )
   END_RUNG
   RUNG wire#powerrail
      Contact( #AreaInterface.Man )
      I_Contact( #CIn.Manager.Control_ON )
      Contact( #Sts.OP_PCoda_CanMoveFreely )
   END_RUNG wire#w1
   RUNG wire#powerrail
      Contact( #CIn.Manager.BattutaVrt.Work )
      wire#w2
      Coil( #Sts.BattutaVrt.Op_Work_Cnd )
   END_RUNG
   RUNG wire#powerrail
      Contact( #AreaInterface.Man )
      I_Contact( #CIn.Manager.Control_ON )
      Contact( #Sts.OP_PCoda_CanMoveFreely )
   END_RUNG wire#w2
   // the same network as SCL:
   #Sts.BattutaVrt.OP_Rest_Cnd := #CIn.Manager.BattutaVrt.Rest OR (#AreaInterface.Man AND NOT #CIn.Manager.Control_ON AND #Sts.OP_PCoda_CanMoveFreely);
   #Sts.BattutaVrt.Op_Work_Cnd := #CIn.Manager.BattutaVrt.Work OR (#AreaInterface.Man AND NOT #CIn.Manager.Control_ON AND #Sts.OP_PCoda_CanMoveFreely);
END_REGION

REGION Network 28: [Paregg Long] - Condizioni movimento Operazione a Lavoro / Riposo
   RUNG wire#powerrail
      Contact( #CIn.Manager.PareggLong.Rest )
      wire#w1
      Coil( #Sts.PareggLong.OP_Rest_Cnd )
   END_RUNG
   RUNG wire#powerrail
      Contact( #AreaInterface.Man )
      I_Contact( #CIn.Manager.Control_ON )
      Contact( #Sts.OP_PCoda_CanMoveFreely )
   END_RUNG wire#w1
   RUNG wire#powerrail
      Contact( #CIn.Manager.PareggLong.Work )
      wire#w2
      Coil( #Sts.PareggLong.Op_Work_Cnd )
   END_RUNG
   RUNG wire#powerrail
      Contact( #AreaInterface.Man )
      I_Contact( #CIn.Manager.Control_ON )
      Contact( #Sts.OP_PCoda_CanMoveFreely )
   END_RUNG wire#w2
   // the same network as SCL:
   #Sts.PareggLong.OP_Rest_Cnd := #CIn.Manager.PareggLong.Rest OR (#AreaInterface.Man AND NOT #CIn.Manager.Control_ON AND #Sts.OP_PCoda_CanMoveFreely);
   #Sts.PareggLong.Op_Work_Cnd := #CIn.Manager.PareggLong.Work OR (#AreaInterface.Man AND NOT #CIn.Manager.Control_ON AND #Sts.OP_PCoda_CanMoveFreely);
END_REGION

REGION Network 29: <+>
END_REGION

REGION Network 30 (SCL): Carro Pareggiatore di Coda - CIn Abilitazioni Stop Manager
   #PareggiatoreLong.Cin.Manager.EnableStopDoorOpeningReq := #BattutaVerticale.Cin.Manager.EnableStopDoorOpeningReq
   := #Bloccaggio.Cin.Manager.EnableStopDoorOpeningReq := #Ax.CIn.Manager.EnableStopDoorOpeningReq := #CIn.Manager.EnableStopDoorOpeningReq;

   #PareggiatoreLong.Cin.Manager.EnableStopInPhase := #BattutaVerticale.Cin.Manager.EnableStopInPhase
   := #Bloccaggio.Cin.Manager.EnableStopInPhase := #Ax.CIn.Manager.EnableStopInPhase := #CIn.Manager.EnableStopInPhase;

   #PareggiatoreLong.Cin.Manager.EnableStopProgrammed := #BattutaVerticale.Cin.Manager.EnableStopProgrammed
   := #Bloccaggio.Cin.Manager.EnableStopProgrammed := #Ax.CIn.Manager.EnableStopProgrammed := #CIn.Manager.EnableStopProgrammed;
END_REGION

REGION Network 31: <+>
END_REGION

REGION Network 32: <<< BLOCCAGGIO SU CREMAGLIERA >>>
END_REGION

REGION Network 33: [Bloccaggio] - Cin Manager (Esecuzione sequenza comandi)
   RUNG wire#powerrail
      I_Contact( #CIn.SemiAut_Pb )
      I_Contact( #AreaInterface.Cycle )
      Not()
      wire#w1
      Contact( #Ctrl.Ax.OP_MoveToPos )
      I_Contact( #COut.Ax_InWPos )
      wire#w2
      Coil( #Bloccaggio.Cin.Manager.Rest )
   END_RUNG
   RUNG wire#w1
      Contact( #CIn.Manager.Bloccaggio.Rest )
   END_RUNG wire#w2
   RUNG wire#w1
      Contact( #Par.Bloccaggio_Sens."2191B1".Enable )
      I_Contact( #Alarm.Bloccaggio_AnalSens_Issue )
      Contact( #Bloccaggio_AnalSens.Q )
      wire#w3
      Contact( #COut.Ax_InWPos )
      Contact( #Ax.COut.Standstill )
      Coil( #Bloccaggio.Cin.Manager.Work )
   END_RUNG
   RUNG wire#w1
      Contact( #CIn.Manager.Bloccaggio.Work )
   END_RUNG wire#w3
   RUNG wire#w1
      I_Contact( #Par.Bloccaggio_Sens."2191B1".Enable )
   END_RUNG wire#w3
   // the same network as SCL:
   #_w1 := NOT (NOT #CIn.SemiAut_Pb AND NOT #AreaInterface.Cycle);
   #Bloccaggio.Cin.Manager.Rest := #_w1 AND ((#Ctrl.Ax.OP_MoveToPos AND NOT #COut.Ax_InWPos) OR #CIn.Manager.Bloccaggio.Rest);
   #Bloccaggio.Cin.Manager.Work := #_w1 AND ((#Par.Bloccaggio_Sens."2191B1".Enable AND NOT #Alarm.Bloccaggio_AnalSens_Issue AND #Bloccaggio_AnalSens.Q) OR #CIn.Manager.Bloccaggio.Work OR NOT #Par.Bloccaggio_Sens."2191B1".Enable) AND #COut.Ax_InWPos AND #Ax.COut.Standstill;
END_REGION

REGION Network 34: [Bloccaggio] - CIn External Alarm
   RUNG wire#powerrail
      Contact( FALSE )
      Coil( #Bloccaggio.Cin.ExternalAlarms )
   END_RUNG
   // the same network as SCL:
   #Bloccaggio.Cin.ExternalAlarms := FALSE;
END_REGION

REGION Network 35: [Bloccaggio] - CIn External Enable
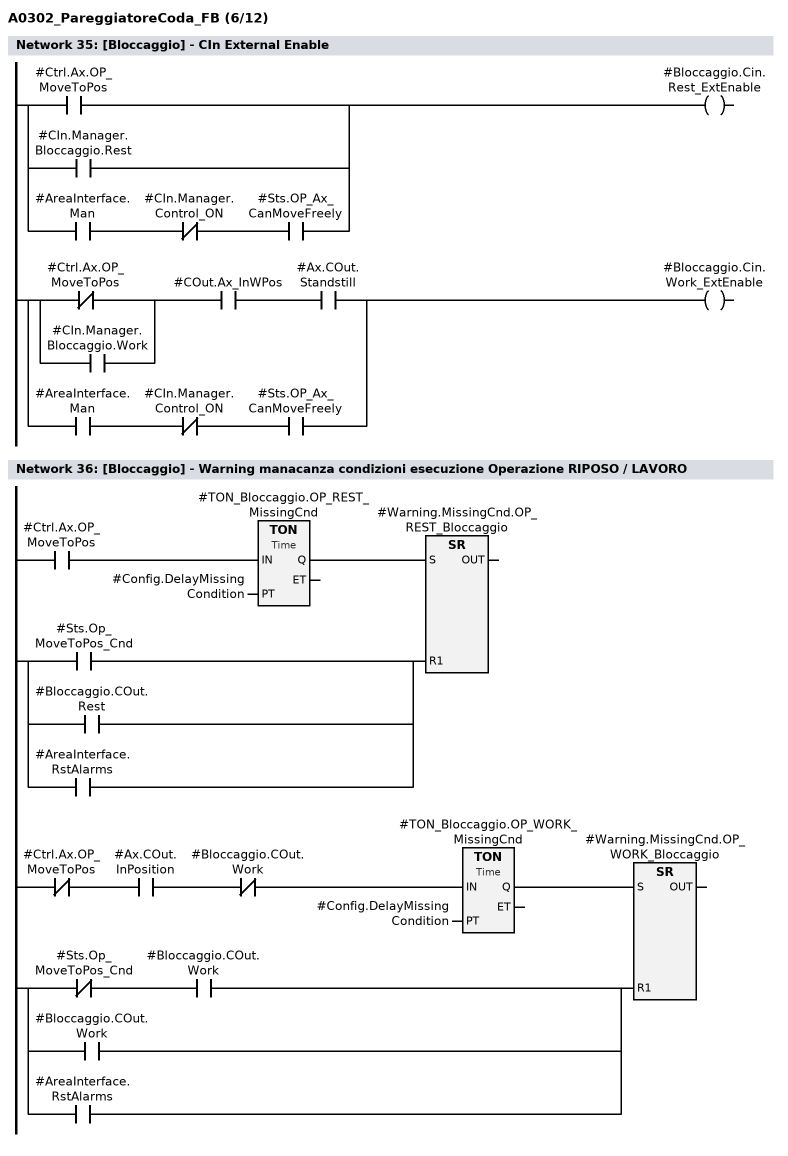
   RUNG wire#powerrail
      Contact( #Ctrl.Ax.OP_MoveToPos )
      wire#w1
      Coil( #Bloccaggio.Cin.Rest_ExtEnable )
   END_RUNG
   RUNG wire#powerrail
      Contact( #CIn.Manager.Bloccaggio.Rest )
   END_RUNG wire#w1
   RUNG wire#powerrail
      Contact( #AreaInterface.Man )
      I_Contact( #CIn.Manager.Control_ON )
      Contact( #Sts.OP_Ax_CanMoveFreely )
   END_RUNG wire#w1
   RUNG wire#powerrail
      I_Contact( #Ctrl.Ax.OP_MoveToPos )
      wire#w2
      Contact( #COut.Ax_InWPos )
      Contact( #Ax.COut.Standstill )
      wire#w3
      Coil( #Bloccaggio.Cin.Work_ExtEnable )
   END_RUNG
   RUNG wire#powerrail
      Contact( #CIn.Manager.Bloccaggio.Work )
   END_RUNG wire#w2
   RUNG wire#powerrail
      Contact( #AreaInterface.Man )
      I_Contact( #CIn.Manager.Control_ON )
      Contact( #Sts.OP_Ax_CanMoveFreely )
   END_RUNG wire#w3
   // the same network as SCL:
   #Bloccaggio.Cin.Rest_ExtEnable := #Ctrl.Ax.OP_MoveToPos OR #CIn.Manager.Bloccaggio.Rest OR (#AreaInterface.Man AND NOT #CIn.Manager.Control_ON AND #Sts.OP_Ax_CanMoveFreely);
   #Bloccaggio.Cin.Work_ExtEnable := ((NOT #Ctrl.Ax.OP_MoveToPos OR #CIn.Manager.Bloccaggio.Work) AND #COut.Ax_InWPos AND #Ax.COut.Standstill) OR (#AreaInterface.Man AND NOT #CIn.Manager.Control_ON AND #Sts.OP_Ax_CanMoveFreely);
END_REGION

REGION Network 36: [Bloccaggio] - Warning manacanza condizioni esecuzione Operazione RIPOSO / LAVORO
   RUNG wire#powerrail
      Contact( #Ctrl.Ax.OP_MoveToPos )
      { S7_Templates := "time_type := Time" } #TON_Bloccaggio.OP_REST_MissingCnd.TON(pt := #Config.DelayMissingCondition, et =>)
      S_SR(operand := #Warning.MissingCnd.OP_REST_Bloccaggio, r1 := wire#w1)
   END_RUNG
   RUNG wire#powerrail
      Contact( #Sts.Op_MoveToPos_Cnd )
   END_RUNG wire#w1
   RUNG wire#powerrail
      Contact( #Bloccaggio.COut.Rest )
   END_RUNG wire#w1
   RUNG wire#powerrail
      Contact( #AreaInterface.RstAlarms )
   END_RUNG wire#w1
   RUNG wire#powerrail
      I_Contact( #Ctrl.Ax.OP_MoveToPos )
      Contact( #Ax.COut.InPosition )
      I_Contact( #Bloccaggio.COut.Work )
      { S7_Templates := "time_type := Time" } #TON_Bloccaggio.OP_WORK_MissingCnd.TON(pt := #Config.DelayMissingCondition, et =>)
      S_SR(operand := #Warning.MissingCnd.OP_WORK_Bloccaggio, r1 := wire#w2)
   END_RUNG
   RUNG wire#powerrail
      I_Contact( #Sts.Op_MoveToPos_Cnd )
      Contact( #Bloccaggio.COut.Work )
   END_RUNG wire#w2
   RUNG wire#powerrail
      Contact( #Bloccaggio.COut.Work )
   END_RUNG wire#w2
   RUNG wire#powerrail
      Contact( #AreaInterface.RstAlarms )
   END_RUNG wire#w2
   // the same network as SCL:
   #TON_Bloccaggio.OP_REST_MissingCnd.TON(IN := #Ctrl.Ax.OP_MoveToPos, PT := #Config.DelayMissingCondition);
   IF #TON_Bloccaggio.OP_REST_MissingCnd.Q THEN
       #Warning.MissingCnd.OP_REST_Bloccaggio := TRUE;   // SR flip-flop
   END_IF;
   IF #Sts.Op_MoveToPos_Cnd OR #Bloccaggio.COut.Rest OR #AreaInterface.RstAlarms THEN
       #Warning.MissingCnd.OP_REST_Bloccaggio := FALSE;
   END_IF;
   #TON_Bloccaggio.OP_WORK_MissingCnd.TON(IN := NOT #Ctrl.Ax.OP_MoveToPos AND #Ax.COut.InPosition AND NOT #Bloccaggio.COut.Work,
                           PT := #Config.DelayMissingCondition);
   IF #TON_Bloccaggio.OP_WORK_MissingCnd.Q THEN
       #Warning.MissingCnd.OP_WORK_Bloccaggio := TRUE;   // SR flip-flop
   END_IF;
   IF (NOT #Sts.Op_MoveToPos_Cnd AND #Bloccaggio.COut.Work) OR #Bloccaggio.COut.Work OR #AreaInterface.RstAlarms THEN
       #Warning.MissingCnd.OP_WORK_Bloccaggio := FALSE;
   END_IF;
END_REGION

REGION Network 37: [Bloccaggio] - Sensore controllo pressione a lavoro su cremaliera
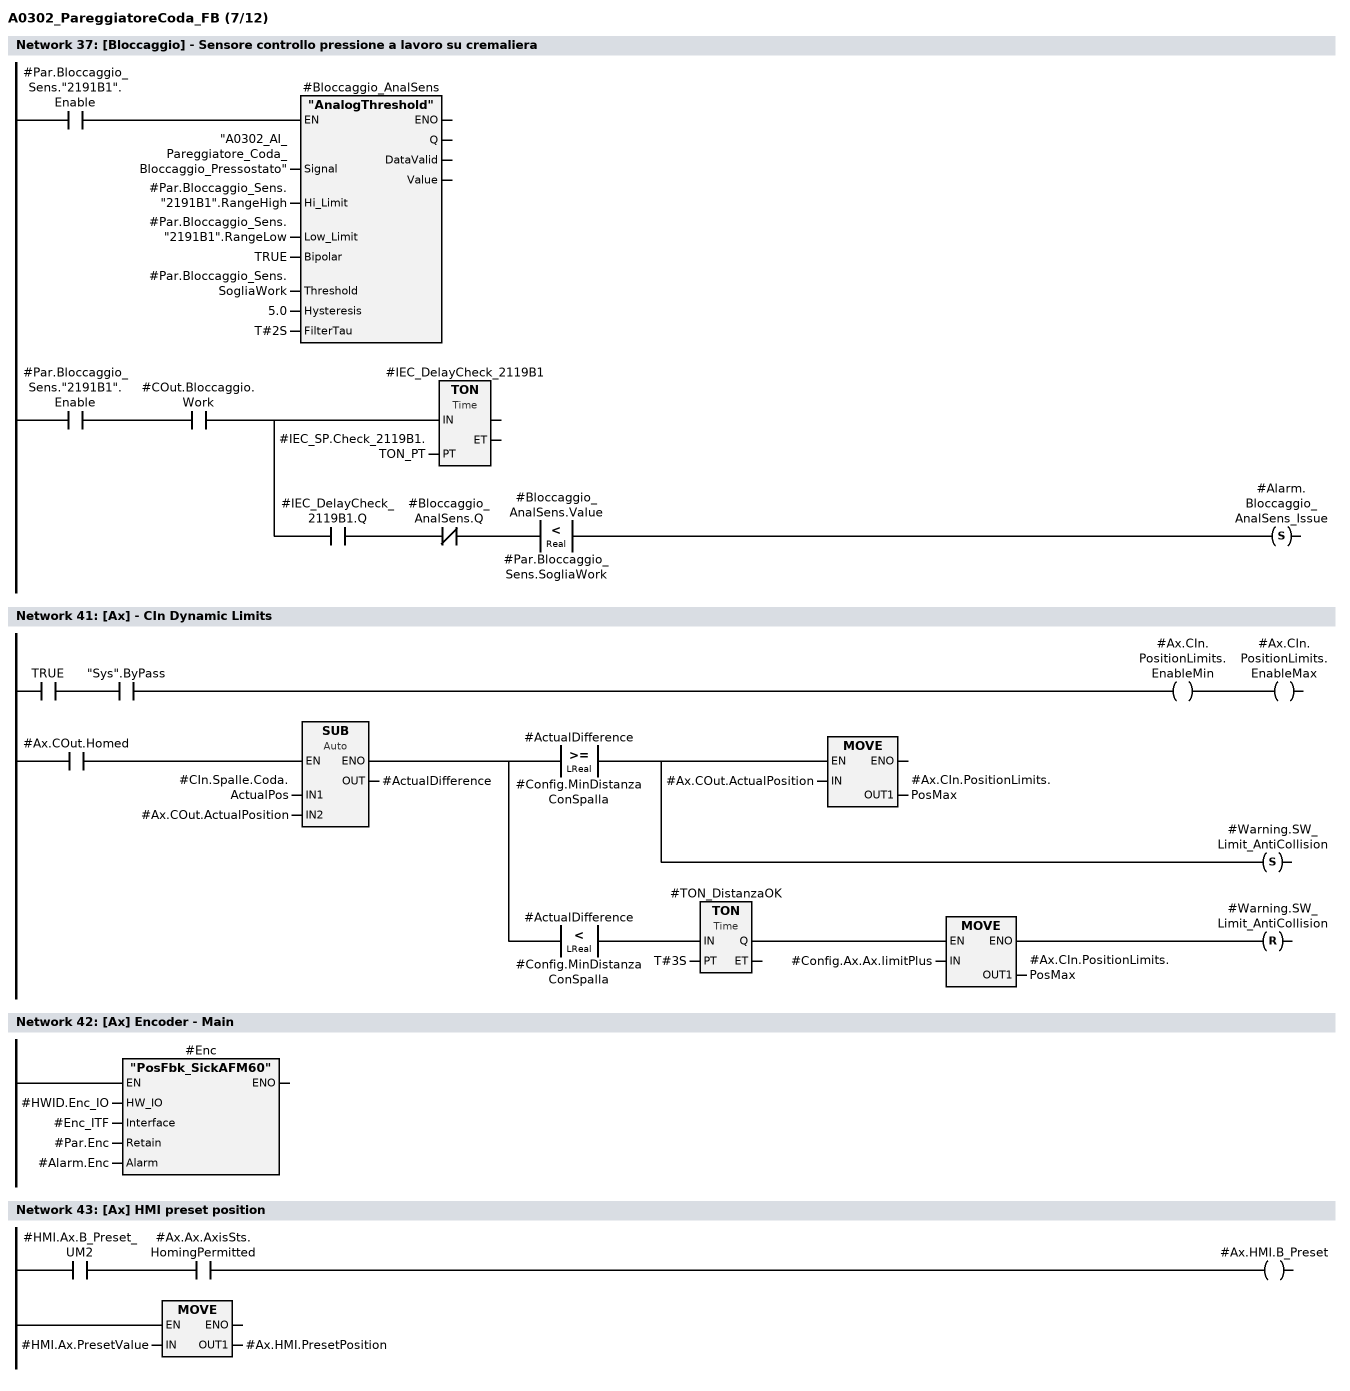
   RUNG wire#powerrail
      Contact( #Par.Bloccaggio_Sens."2191B1".Enable )
      #Bloccaggio_AnalSens(Signal := "A0302_AI_Pareggiatore_Coda_Bloccaggio_Pressostato", Hi_Limit := #Par.Bloccaggio_Sens."2191B1".RangeHigh, Low_Limit := #Par.Bloccaggio_Sens."2191B1".RangeLow, Bipolar := TRUE, Threshold := #Par.Bloccaggio_Sens.SogliaWork, Hysteresis := 5.0, FilterTau := T#2S, Q =>, DataValid =>, Value =>)
   END_RUNG
   RUNG wire#powerrail
      Contact( #Par.Bloccaggio_Sens."2191B1".Enable )
      Contact( #COut.Bloccaggio.Work )
      wire#w1
      { S7_Templates := "time_type := Time" } #IEC_DelayCheck_2119B1.TON(pt := #IEC_SP.Check_2119B1.TON_PT, et =>)
   END_RUNG
   RUNG wire#w1
      Contact( #IEC_DelayCheck_2119B1.Q )
      I_Contact( #Bloccaggio_AnalSens.Q )
      { S7_Templates := "SrcType := Real" } LT_Contact(in1 := #Bloccaggio_AnalSens.Value, in2 := #Par.Bloccaggio_Sens.SogliaWork)
      S_Coil( #Alarm.Bloccaggio_AnalSens_Issue )
   END_RUNG
   // the same network as SCL:
   IF #Par.Bloccaggio_Sens."2191B1".Enable THEN
       #Bloccaggio_AnalSens(Signal := "A0302_AI_Pareggiatore_Coda_Bloccaggio_Pressostato",   // "AnalogThreshold"
                            Hi_Limit := #Par.Bloccaggio_Sens."2191B1".RangeHigh,
                            Low_Limit := #Par.Bloccaggio_Sens."2191B1".RangeLow,
                            Bipolar := TRUE,
                            Threshold := #Par.Bloccaggio_Sens.SogliaWork,
                            Hysteresis := 5.0,
                            FilterTau := T#2S);
   END_IF;
   #_w1 := #Par.Bloccaggio_Sens."2191B1".Enable AND #COut.Bloccaggio.Work;
   #IEC_DelayCheck_2119B1.TON(IN := #_w1, PT := #IEC_SP.Check_2119B1.TON_PT);
   IF #_w1 AND #IEC_DelayCheck_2119B1.Q AND NOT #Bloccaggio_AnalSens.Q AND (#Bloccaggio_AnalSens.Value < #Par.Bloccaggio_Sens.SogliaWork) THEN
       #Alarm.Bloccaggio_AnalSens_Issue := TRUE;
   END_IF;
END_REGION

REGION Network 39 (SCL): == Calcolo setpoint posizione carri in funzione della cremaliera in Manuale ==
   // Foglio di calcolo posizione Cremaliera fornito
   // 
   IF #AreaInterface.Man AND #Ctrl.Ax.OP_MoveToPos THEN

       #CarroCoda.PosBattutePz := (#Par.CarroPareggCoda.Preset - "A0302_PareggiatoreCoda_PERS".Par_Sens.AI.RangeLow);
       #CarroCoda.RimanenzaPos := (#Ax.HMI.TargetPosition - #Ax.Ctrl.Pos - #CarroCoda.PosBattutePz) + ("A0302_PareggiatoreCoda_PERS".Par_Sens.AI.RangeLow + 2.0);
       #CarroCoda.NrPassiReq := (#CarroCoda.RimanenzaPos / #Par.Cremaliera.Passo);

       // Calcolo i numeri di passi cremaliera richiesti per spostarmi della rimanenza
       #CarroCoda.PassoReq := ROUND(#CarroCoda.NrPassiReq);

       #Ax.Ctrl.Pos := (#CarroCoda.PassoReq * #Par.Cremaliera.Passo) + #CarroCoda.PosBattutePz + "A0302_PareggiatoreCoda_PERS".Par_Sens.AI.RangeLow;

   END_IF;


       (*
       // Calcolo la rimanenza dello spazio tra lo 0 e il preset dei carri
       #CarroCoda.RimanenzaPos := #Ax.HMI.TargetPosition - #Par.CarroPareggCoda.Preset;

       // Calcolo i numeri di passi cremaliera richiesti per spostarmi della rimanenza
       #CarroCoda.PassoReq := ROUND(#CarroCoda.RimanenzaPos / #Par.Cremaliera.Passo);

       // Calcolo del setpoint di posizione dei 2 carri in funzione della misura calcolata - Se cambia il Beam Len viene richiesto il nuovo riposizionamento
       #Ax.Ctrl.Pos := (#CarroCoda.PassoReq * #Par.Cremaliera.Passo) + #Par.CarroPareggCoda.Preset;
   END_IF;
   *)
END_REGION

REGION Network 40: <<< AXIS >>>
END_REGION

REGION Network 41: [Ax] - CIn Dynamic Limits
   RUNG wire#powerrail
      Contact( TRUE )
      Contact( "Sys".ByPass )
      Coil( #Ax.CIn.PositionLimits.EnableMin )
      Coil( #Ax.CIn.PositionLimits.EnableMax )
   END_RUNG
   RUNG wire#powerrail
      Contact( #Ax.COut.Homed )
      Sub(in1 := #CIn.Spalle.Coda.ActualPos, in2 := #Ax.COut.ActualPosition, out => #ActualDifference)
      wire#w1
      { S7_Templates := "SrcType := LReal" } GE_Contact(in1 := #ActualDifference, in2 := #Config.MinDistanzaConSpalla)
      wire#w2
      Move(in := #Ax.COut.ActualPosition, out1 => #Ax.CIn.PositionLimits.PosMax)
   END_RUNG
   RUNG wire#w2
      S_Coil( #Warning.SW_Limit_AntiCollision )
   END_RUNG
   RUNG wire#w1
      { S7_Templates := "SrcType := LReal" } LT_Contact(in1 := #ActualDifference, in2 := #Config.MinDistanzaConSpalla)
      { S7_Templates := "time_type := Time" } #TON_DistanzaOK.TON(pt := T#3S, et =>)
      Move(in := #Config.Ax.Ax.limitPlus, out1 => #Ax.CIn.PositionLimits.PosMax)
      R_Coil( #Warning.SW_Limit_AntiCollision )
   END_RUNG
   // the same network as SCL:
   #Ax.CIn.PositionLimits.EnableMin := TRUE AND "Sys".ByPass;
   #Ax.CIn.PositionLimits.EnableMax := #Ax.CIn.PositionLimits.EnableMin;
   IF #Ax.COut.Homed THEN #ActualDifference := #CIn.Spalle.Coda.ActualPos - #Ax.COut.ActualPosition; END_IF;
   IF #Ax.COut.Homed AND (#ActualDifference >= #Config.MinDistanzaConSpalla) THEN
       #Ax.CIn.PositionLimits.PosMax := #Ax.COut.ActualPosition;
       #Warning.SW_Limit_AntiCollision := TRUE;
   END_IF;
   #TON_DistanzaOK.TON(IN := #Ax.COut.Homed AND (#ActualDifference < #Config.MinDistanzaConSpalla), PT := T#3S);
   IF #TON_DistanzaOK.Q THEN
       #Ax.CIn.PositionLimits.PosMax := #Config.Ax.Ax.limitPlus;
       #Warning.SW_Limit_AntiCollision := FALSE;
   END_IF;
END_REGION

REGION Network 42: [Ax] Encoder - Main
   RUNG wire#powerrail
      #Enc(HW_IO := #HWID.Enc_IO, Interface := #Enc_ITF, Retain := #Par.Enc, Alarm := #Alarm.Enc)
   END_RUNG
   // the same network as SCL:
   #Enc(HW_IO := #HWID.Enc_IO, Interface := #Enc_ITF, Retain := #Par.Enc, Alarm := #Alarm.Enc);   // "PosFbk_SickAFM60"
END_REGION

REGION Network 43: [Ax] HMI preset position
   RUNG wire#powerrail
      Contact( #HMI.Ax.B_Preset_UM2 )
      Contact( #Ax.Ax.AxisSts.HomingPermitted )
      Coil( #Ax.HMI.B_Preset )
   END_RUNG
   RUNG wire#powerrail
      Move(in := #HMI.Ax.PresetValue, out1 => #Ax.HMI.PresetPosition)
   END_RUNG
   // the same network as SCL:
   #Ax.HMI.B_Preset := #HMI.Ax.B_Preset_UM2 AND #Ax.Ax.AxisSts.HomingPermitted;
   #Ax.HMI.PresetPosition := #HMI.Ax.PresetValue;
END_REGION

REGION Network 44: [Ax] - CIn External Enable
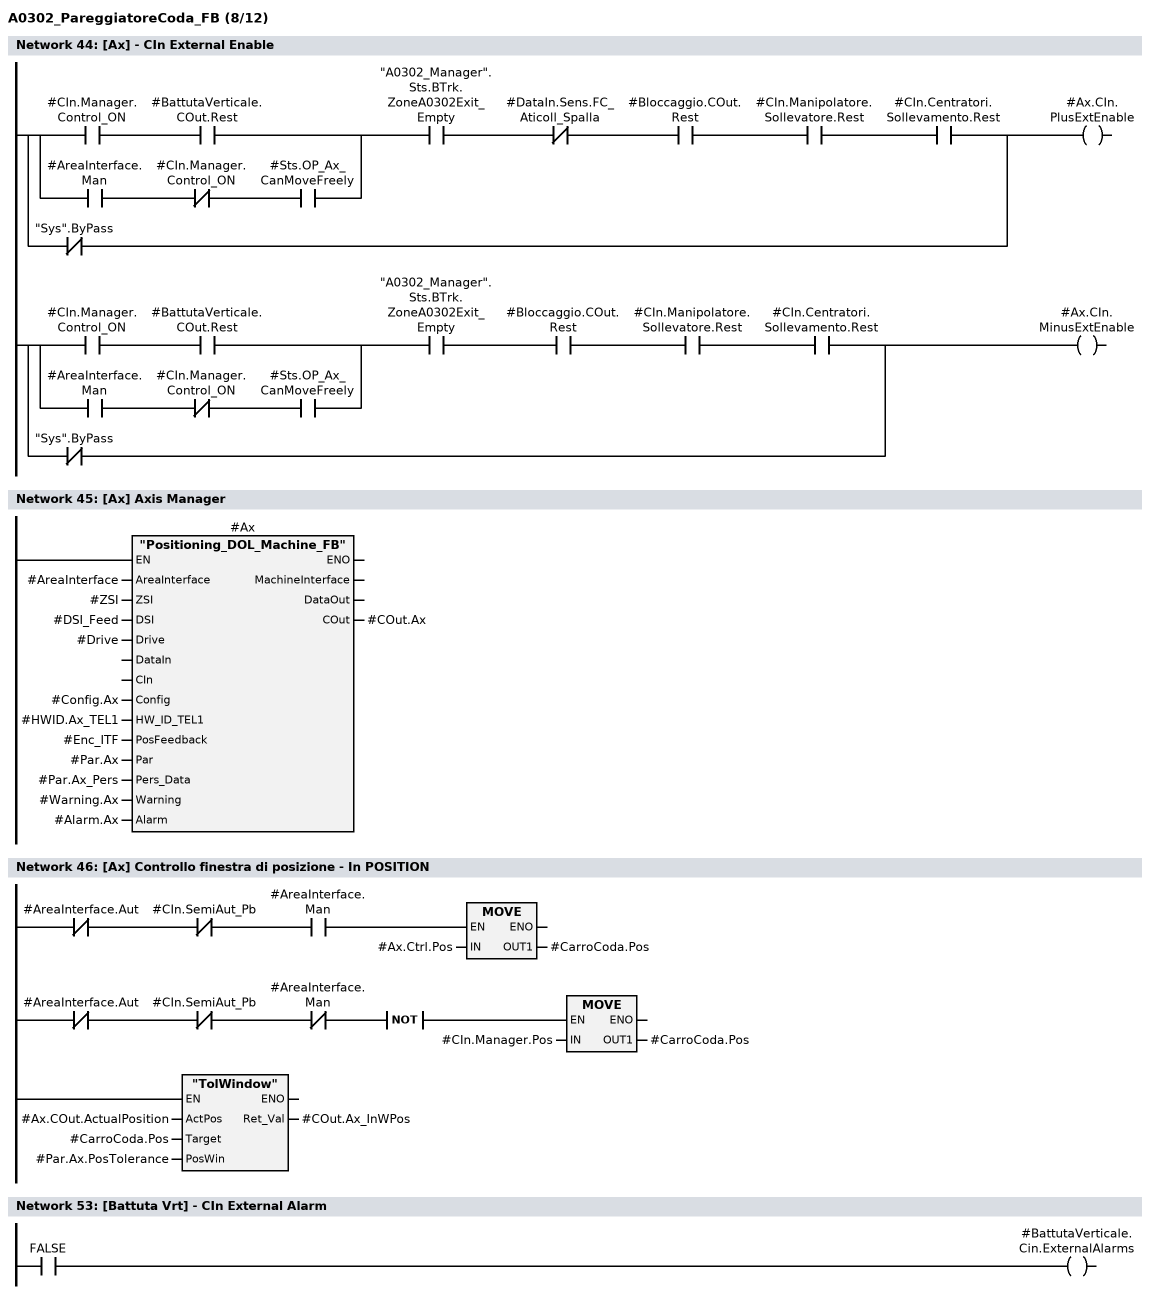
   RUNG wire#powerrail
      Contact( #CIn.Manager.Control_ON )
      Contact( #BattutaVerticale.COut.Rest )
      wire#w1
      Contact( "A0302_Manager".Sts.BTrk.ZoneA0302Exit_Empty )
      I_Contact( #DataIn.Sens.FC_Aticoll_Spalla )
      Contact( #Bloccaggio.COut.Rest )
      Contact( #CIn.Manipolatore.Sollevatore.Rest )
      Contact( #CIn.Centratori.Sollevamento.Rest )
      wire#w2
      Coil( #Ax.CIn.PlusExtEnable )
   END_RUNG
   RUNG wire#powerrail
      Contact( #AreaInterface.Man )
      I_Contact( #CIn.Manager.Control_ON )
      Contact( #Sts.OP_Ax_CanMoveFreely )
   END_RUNG wire#w1
   RUNG wire#powerrail
      I_Contact( "Sys".ByPass )
   END_RUNG wire#w2
   RUNG wire#powerrail
      Contact( #CIn.Manager.Control_ON )
      Contact( #BattutaVerticale.COut.Rest )
      wire#w3
      Contact( "A0302_Manager".Sts.BTrk.ZoneA0302Exit_Empty )
      Contact( #Bloccaggio.COut.Rest )
      Contact( #CIn.Manipolatore.Sollevatore.Rest )
      Contact( #CIn.Centratori.Sollevamento.Rest )
      wire#w4
      Coil( #Ax.CIn.MinusExtEnable )
   END_RUNG
   RUNG wire#powerrail
      Contact( #AreaInterface.Man )
      I_Contact( #CIn.Manager.Control_ON )
      Contact( #Sts.OP_Ax_CanMoveFreely )
   END_RUNG wire#w3
   RUNG wire#powerrail
      I_Contact( "Sys".ByPass )
   END_RUNG wire#w4
   // the same network as SCL:
   #Ax.CIn.PlusExtEnable := (((#CIn.Manager.Control_ON AND #BattutaVerticale.COut.Rest) OR (#AreaInterface.Man AND NOT #CIn.Manager.Control_ON AND #Sts.OP_Ax_CanMoveFreely)) AND "A0302_Manager".Sts.BTrk.ZoneA0302Exit_Empty AND NOT #DataIn.Sens.FC_Aticoll_Spalla AND #Bloccaggio.COut.Rest AND #CIn.Manipolatore.Sollevatore.Rest AND #CIn.Centratori.Sollevamento.Rest) OR NOT "Sys".ByPass;
   #Ax.CIn.MinusExtEnable := (((#CIn.Manager.Control_ON AND #BattutaVerticale.COut.Rest) OR (#AreaInterface.Man AND NOT #CIn.Manager.Control_ON AND #Sts.OP_Ax_CanMoveFreely)) AND "A0302_Manager".Sts.BTrk.ZoneA0302Exit_Empty AND #Bloccaggio.COut.Rest AND #CIn.Manipolatore.Sollevatore.Rest AND #CIn.Centratori.Sollevamento.Rest) OR NOT "Sys".ByPass;
END_REGION

REGION Network 45: [Ax] Axis Manager
   RUNG wire#powerrail
      #Ax(AreaInterface := #AreaInterface, ZSI := #ZSI, DSI := #DSI_Feed, Drive := #Drive, DataIn :=, CIn :=, Config := #Config.Ax, HW_ID_TEL1 := #HWID.Ax_TEL1, PosFeedback := #Enc_ITF, Par := #Par.Ax, Pers_Data := #Par.Ax_Pers, Warning := #Warning.Ax, Alarm := #Alarm.Ax, MachineInterface =>, DataOut =>, COut => #COut.Ax)
   END_RUNG
   // the same network as SCL:
   #Ax(AreaInterface := #AreaInterface,   // "Positioning_DOL_Machine_FB"
       ZSI := #ZSI,
       DSI := #DSI_Feed,
       Drive := #Drive,
       Config := #Config.Ax,
       HW_ID_TEL1 := #HWID.Ax_TEL1,
       PosFeedback := #Enc_ITF,
       Par := #Par.Ax,
       Pers_Data := #Par.Ax_Pers,
       Warning := #Warning.Ax,
       Alarm := #Alarm.Ax,
       COut => #COut.Ax);
END_REGION

REGION Network 46: [Ax] Controllo finestra di posizione - In POSITION
   RUNG wire#powerrail
      I_Contact( #AreaInterface.Aut )
      I_Contact( #CIn.SemiAut_Pb )
      Contact( #AreaInterface.Man )
      Move(in := #Ax.Ctrl.Pos, out1 => #CarroCoda.Pos)
   END_RUNG
   RUNG wire#powerrail
      I_Contact( #AreaInterface.Aut )
      I_Contact( #CIn.SemiAut_Pb )
      I_Contact( #AreaInterface.Man )
      Not()
      Move(in := #CIn.Manager.Pos, out1 => #CarroCoda.Pos)
   END_RUNG
   RUNG wire#powerrail
      "TolWindow"(ActPos := #Ax.COut.ActualPosition, Target := #CarroCoda.Pos, PosWin := #Par.Ax.PosTolerance, Ret_Val => #COut.Ax_InWPos)
   END_RUNG
   // the same network as SCL:
   IF NOT #AreaInterface.Aut AND NOT #CIn.SemiAut_Pb AND #AreaInterface.Man THEN
       #CarroCoda.Pos := #Ax.Ctrl.Pos;
   END_IF;
   IF NOT (NOT #AreaInterface.Aut AND NOT #CIn.SemiAut_Pb AND NOT #AreaInterface.Man) THEN
       #CarroCoda.Pos := #CIn.Manager.Pos;
   END_IF;
   #COut.Ax_InWPos := "TolWindow"(ActPos := #Ax.COut.ActualPosition,
                           Target := #CarroCoda.Pos,
                           PosWin := #Par.Ax.PosTolerance);
END_REGION

REGION Network 47 (SCL): [Ax] - Cin Manager (Esecuzione sequenza comandi)
   // Operazione LAVORO dell' asse spintore quando i 2 ciclindri sono in riposo e il bloccaggio è a riposo
   #Ax.CIn.Manager.Control_ON := #Ax.DSI.PowerEnable := #Bloccaggio.Cin.Manager.Control_ON  := #Ctrl.Ax.OP_MoveToPos AND NOT #DataIn.Sens.FC_Aticoll_Spalla;



   IF #Ctrl.Ax.OP_MoveToPos AND #Sts.Op_MoveToPos_Cnd AND NOT #COut.Ax_InWPos AND #Bloccaggio.COut.Rest
           AND #BattutaVerticale.Cin.Manager.Rest AND #PareggiatoreLong.Cin.Manager.Rest THEN
           #Ax.CIn.Manager.MoveToPos := TRUE;

           // Se raggiungo la posizione di setpoint spengo il comando
       ELSIF #COut.Ax_InWPos AND #Ax.COut.Standstill THEN
           #Ax.CIn.Manager.MoveToPos := FALSE;
           #Ax.DSI.PowerEnable := FALSE;
       END_IF;

   // Attivazione ALLARME collisione con spalla
   // 
       IF #Ax.CIn.Manager.Control_ON AND #Ax.CIn.Manager.MoveToPos AND #DataIn.Sens.FC_Aticoll_Spalla THEN

           #Alarm.SensFC_Aticoll_Spalla := TRUE;
           #Ax.CIn.Manager.MoveToPos := FALSE;
           #Ax.DSI.PowerEnable := FALSE;
       END_IF;
END_REGION

REGION Network 48: <+>
END_REGION

REGION Network 49 (SCL): [Battuta Vrt ] - Cin Manager (Esecuzione sequenza comandi)
   // Comando CIn Manager ControlON di tutte le utenze
   #BattutaVerticale.Cin.Manager.Control_ON := #CIn.Manager.Control_ON;

   #BattutaVerticale.Cin.Manager.Rest := FALSE;
   #BattutaVerticale.Cin.Manager.Work := FALSE;

   // Gestione dei comandi relativi a Battuta VRT in sequenza quando ho un OP cnd

   IF (#Ctrl.BattutaVrt.OP_Rest AND #Sts.BattutaVrt.OP_Rest_Cnd) OR (#Ctrl.Ax.OP_MoveToPos AND #Sts.Op_MoveToPos_Cnd) THEN

           #PareggiatoreLong.Cin.Manager.Rest := TRUE;
           #BattutaVerticale.Cin.Manager.Rest := #PareggiatoreLong.COut.Rest;

           // Vado a lavoro solo se sono in posizione e il carro è bloccato sulla cremaliera e i pezzi sono centrati sulla rulliera     
       ELSIF  (#Ctrl.BattutaVrt.OP_Work AND #Sts.BattutaVrt.Op_Work_Cnd) AND #Bloccaggio.COut.Work THEN

           #BattutaVerticale.Cin.Manager.Work := TRUE;
           #PareggiatoreLong.Cin.Manager.Rest := NOT #BattutaVerticale.Cin.Manager.Work;

   END_IF;
END_REGION

REGION Network 50 (SCL): [Paregg Long ] - Cin Manager (Esecuzione sequenza comandi)
   // Comando CIn Manager ControlON di tutte le utenze
   #PareggiatoreLong.Cin.Manager.Control_ON := #CIn.Manager.Control_ON;

   #PareggiatoreLong.Cin.Manager.Rest := FALSE;
   #PareggiatoreLong.Cin.Manager.Work := FALSE;

   // Gestione dei comandi relativi a Pareggiatore Longitudinale in sequenza quando ho un OP cnd
   IF (#Ctrl.PareggLong.OP_Rest AND #Sts.PareggLong.OP_Rest_Cnd) OR (#Ctrl.Ax.OP_MoveToPos AND #Sts.Op_MoveToPos_Cnd) THEN

       #PareggiatoreLong.Cin.Manager.Rest := TRUE;
       #PareggiatoreLong.Cin.Manager.Work := FALSE;

           // Vado a lavoro solo se sono in posizione e il carro è bloccato sulla cremaliera e i pezzi sono centrati sulla rulliera     
   ELSIF  (#Ctrl.PareggLong.OP_Work AND #Sts.PareggLong.Op_Work_Cnd) AND #Bloccaggio.COut.Work THEN

           #BattutaVerticale.Cin.Manager.Work := TRUE;
           #PareggiatoreLong.Cin.Manager.Work := #BattutaVerticale.COut.Work;

   END_IF;
END_REGION

REGION Network 51: <+>
END_REGION

REGION Network 52: <<< BATTUTA VERTICALE >>>
END_REGION

REGION Network 53: [Battuta Vrt] - CIn External Alarm
   RUNG wire#powerrail
      Contact( FALSE )
      Coil( #BattutaVerticale.Cin.ExternalAlarms )
   END_RUNG
   // the same network as SCL:
   #BattutaVerticale.Cin.ExternalAlarms := FALSE;
END_REGION

REGION Network 54: [Battuta Vrt] - CIn External Enable
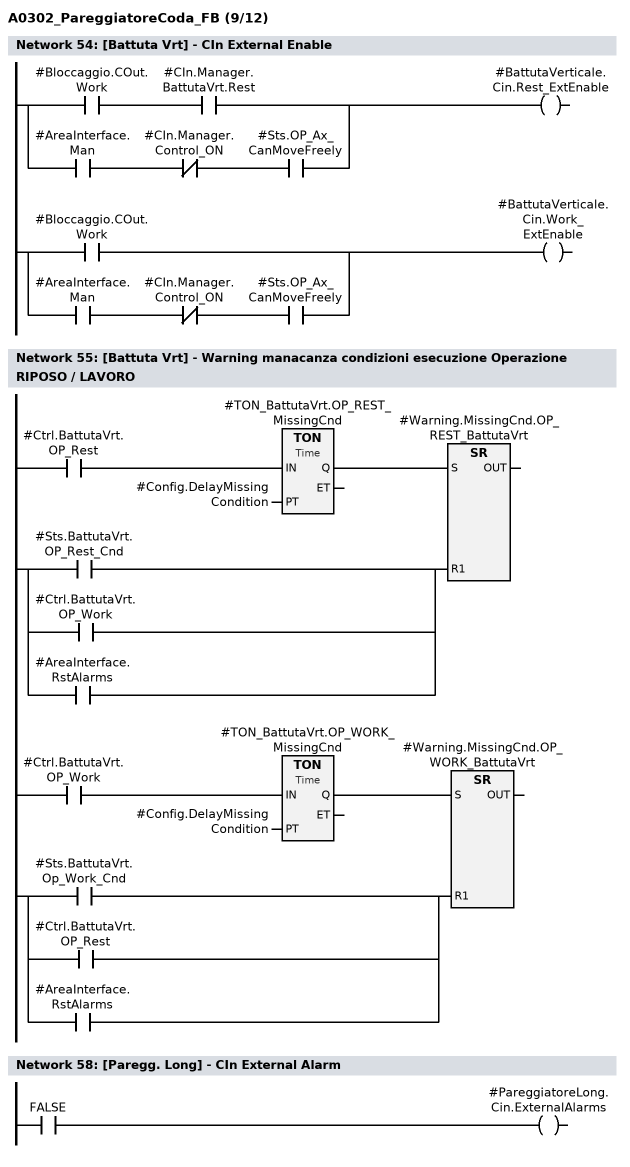
   RUNG wire#powerrail
      Contact( #Bloccaggio.COut.Work )
      Contact( #CIn.Manager.BattutaVrt.Rest )
      wire#w1
      Coil( #BattutaVerticale.Cin.Rest_ExtEnable )
   END_RUNG
   RUNG wire#powerrail
      Contact( #AreaInterface.Man )
      I_Contact( #CIn.Manager.Control_ON )
      Contact( #Sts.OP_Ax_CanMoveFreely )
   END_RUNG wire#w1
   RUNG wire#powerrail
      Contact( #Bloccaggio.COut.Work )
      wire#w2
      Coil( #BattutaVerticale.Cin.Work_ExtEnable )
   END_RUNG
   RUNG wire#powerrail
      Contact( #AreaInterface.Man )
      I_Contact( #CIn.Manager.Control_ON )
      Contact( #Sts.OP_Ax_CanMoveFreely )
   END_RUNG wire#w2
   // the same network as SCL:
   #BattutaVerticale.Cin.Rest_ExtEnable := (#Bloccaggio.COut.Work AND #CIn.Manager.BattutaVrt.Rest) OR (#AreaInterface.Man AND NOT #CIn.Manager.Control_ON AND #Sts.OP_Ax_CanMoveFreely);
   #BattutaVerticale.Cin.Work_ExtEnable := #Bloccaggio.COut.Work OR (#AreaInterface.Man AND NOT #CIn.Manager.Control_ON AND #Sts.OP_Ax_CanMoveFreely);
END_REGION

REGION Network 55: [Battuta Vrt] - Warning manacanza condizioni esecuzione Operazione RIPOSO / LAVORO
   RUNG wire#powerrail
      Contact( #Ctrl.BattutaVrt.OP_Rest )
      { S7_Templates := "time_type := Time" } #TON_BattutaVrt.OP_REST_MissingCnd.TON(pt := #Config.DelayMissingCondition, et =>)
      S_SR(operand := #Warning.MissingCnd.OP_REST_BattutaVrt, r1 := wire#w1)
   END_RUNG
   RUNG wire#powerrail
      Contact( #Sts.BattutaVrt.OP_Rest_Cnd )
   END_RUNG wire#w1
   RUNG wire#powerrail
      Contact( #Ctrl.BattutaVrt.OP_Work )
   END_RUNG wire#w1
   RUNG wire#powerrail
      Contact( #AreaInterface.RstAlarms )
   END_RUNG wire#w1
   RUNG wire#powerrail
      Contact( #Ctrl.BattutaVrt.OP_Work )
      { S7_Templates := "time_type := Time" } #TON_BattutaVrt.OP_WORK_MissingCnd.TON(pt := #Config.DelayMissingCondition, et =>)
      S_SR(operand := #Warning.MissingCnd.OP_WORK_BattutaVrt, r1 := wire#w2)
   END_RUNG
   RUNG wire#powerrail
      Contact( #Sts.BattutaVrt.Op_Work_Cnd )
   END_RUNG wire#w2
   RUNG wire#powerrail
      Contact( #Ctrl.BattutaVrt.OP_Rest )
   END_RUNG wire#w2
   RUNG wire#powerrail
      Contact( #AreaInterface.RstAlarms )
   END_RUNG wire#w2
   // the same network as SCL:
   #TON_BattutaVrt.OP_REST_MissingCnd.TON(IN := #Ctrl.BattutaVrt.OP_Rest, PT := #Config.DelayMissingCondition);
   IF #TON_BattutaVrt.OP_REST_MissingCnd.Q THEN
       #Warning.MissingCnd.OP_REST_BattutaVrt := TRUE;   // SR flip-flop
   END_IF;
   IF #Sts.BattutaVrt.OP_Rest_Cnd OR #Ctrl.BattutaVrt.OP_Work OR #AreaInterface.RstAlarms THEN
       #Warning.MissingCnd.OP_REST_BattutaVrt := FALSE;
   END_IF;
   #TON_BattutaVrt.OP_WORK_MissingCnd.TON(IN := #Ctrl.BattutaVrt.OP_Work, PT := #Config.DelayMissingCondition);
   IF #TON_BattutaVrt.OP_WORK_MissingCnd.Q THEN
       #Warning.MissingCnd.OP_WORK_BattutaVrt := TRUE;   // SR flip-flop
   END_IF;
   IF #Sts.BattutaVrt.Op_Work_Cnd OR #Ctrl.BattutaVrt.OP_Rest OR #AreaInterface.RstAlarms THEN
       #Warning.MissingCnd.OP_WORK_BattutaVrt := FALSE;
   END_IF;
END_REGION

REGION Network 57: <<< PAREGGIATORE LONGITUDINALE >>>
END_REGION

REGION Network 58: [Paregg. Long] - CIn External Alarm
   RUNG wire#powerrail
      Contact( FALSE )
      Coil( #PareggiatoreLong.Cin.ExternalAlarms )
   END_RUNG
   // the same network as SCL:
   #PareggiatoreLong.Cin.ExternalAlarms := FALSE;
END_REGION

REGION Network 59: [Paregg. Long] - CIn External Enable
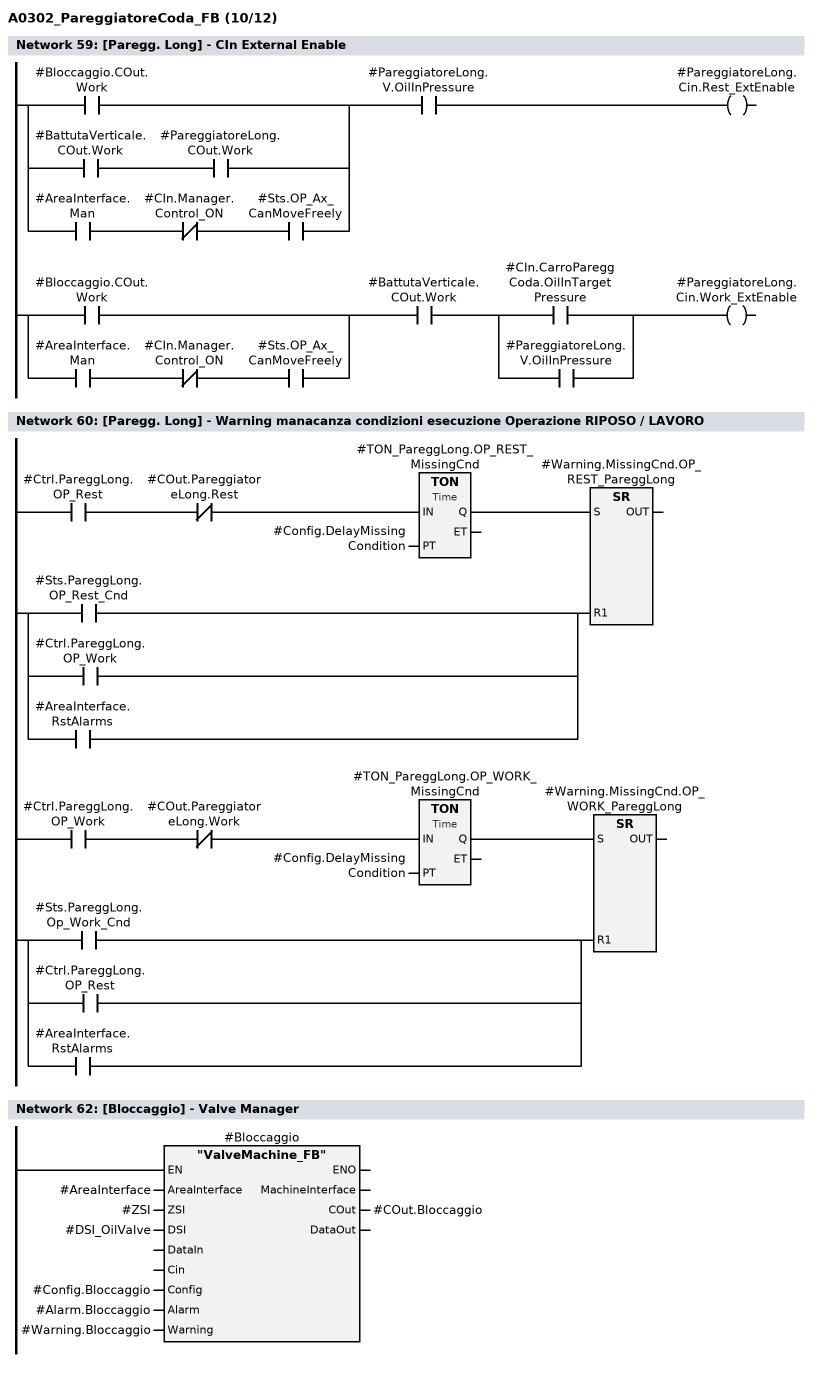
   RUNG wire#powerrail
      Contact( #Bloccaggio.COut.Work )
      wire#w1
      Contact( #PareggiatoreLong.V.OilInPressure )
      Coil( #PareggiatoreLong.Cin.Rest_ExtEnable )
   END_RUNG
   RUNG wire#powerrail
      Contact( #BattutaVerticale.COut.Work )
      Contact( #PareggiatoreLong.COut.Work )
   END_RUNG wire#w1
   RUNG wire#powerrail
      Contact( #AreaInterface.Man )
      I_Contact( #CIn.Manager.Control_ON )
      Contact( #Sts.OP_Ax_CanMoveFreely )
   END_RUNG wire#w1
   RUNG wire#powerrail
      Contact( #Bloccaggio.COut.Work )
      wire#w2
      Contact( #BattutaVerticale.COut.Work )
      wire#w3
      Contact( #CIn.CarroPareggCoda.OilInTargetPressure )
      wire#w4
      Coil( #PareggiatoreLong.Cin.Work_ExtEnable )
   END_RUNG
   RUNG wire#powerrail
      Contact( #AreaInterface.Man )
      I_Contact( #CIn.Manager.Control_ON )
      Contact( #Sts.OP_Ax_CanMoveFreely )
   END_RUNG wire#w2
   RUNG wire#w3
      Contact( #PareggiatoreLong.V.OilInPressure )
   END_RUNG wire#w4
   // the same network as SCL:
   #PareggiatoreLong.Cin.Rest_ExtEnable := (#Bloccaggio.COut.Work OR (#BattutaVerticale.COut.Work AND #PareggiatoreLong.COut.Work) OR (#AreaInterface.Man AND NOT #CIn.Manager.Control_ON AND #Sts.OP_Ax_CanMoveFreely)) AND #PareggiatoreLong.V.OilInPressure;
   #PareggiatoreLong.Cin.Work_ExtEnable := (#Bloccaggio.COut.Work OR (#AreaInterface.Man AND NOT #CIn.Manager.Control_ON AND #Sts.OP_Ax_CanMoveFreely)) AND #BattutaVerticale.COut.Work AND (#CIn.CarroPareggCoda.OilInTargetPressure OR #PareggiatoreLong.V.OilInPressure);
END_REGION

REGION Network 60: [Paregg. Long] - Warning manacanza condizioni esecuzione Operazione RIPOSO / LAVORO
   RUNG wire#powerrail
      Contact( #Ctrl.PareggLong.OP_Rest )
      I_Contact( #COut.PareggiatoreLong.Rest )
      { S7_Templates := "time_type := Time" } #TON_PareggLong.OP_REST_MissingCnd.TON(pt := #Config.DelayMissingCondition, et =>)
      S_SR(operand := #Warning.MissingCnd.OP_REST_PareggLong, r1 := wire#w1)
   END_RUNG
   RUNG wire#powerrail
      Contact( #Sts.PareggLong.OP_Rest_Cnd )
   END_RUNG wire#w1
   RUNG wire#powerrail
      Contact( #Ctrl.PareggLong.OP_Work )
   END_RUNG wire#w1
   RUNG wire#powerrail
      Contact( #AreaInterface.RstAlarms )
   END_RUNG wire#w1
   RUNG wire#powerrail
      Contact( #Ctrl.PareggLong.OP_Work )
      I_Contact( #COut.PareggiatoreLong.Work )
      { S7_Templates := "time_type := Time" } #TON_PareggLong.OP_WORK_MissingCnd.TON(pt := #Config.DelayMissingCondition, et =>)
      S_SR(operand := #Warning.MissingCnd.OP_WORK_PareggLong, r1 := wire#w2)
   END_RUNG
   RUNG wire#powerrail
      Contact( #Sts.PareggLong.Op_Work_Cnd )
   END_RUNG wire#w2
   RUNG wire#powerrail
      Contact( #Ctrl.PareggLong.OP_Rest )
   END_RUNG wire#w2
   RUNG wire#powerrail
      Contact( #AreaInterface.RstAlarms )
   END_RUNG wire#w2
   // the same network as SCL:
   #TON_PareggLong.OP_REST_MissingCnd.TON(IN := #Ctrl.PareggLong.OP_Rest AND NOT #COut.PareggiatoreLong.Rest,
                           PT := #Config.DelayMissingCondition);
   IF #TON_PareggLong.OP_REST_MissingCnd.Q THEN
       #Warning.MissingCnd.OP_REST_PareggLong := TRUE;   // SR flip-flop
   END_IF;
   IF #Sts.PareggLong.OP_Rest_Cnd OR #Ctrl.PareggLong.OP_Work OR #AreaInterface.RstAlarms THEN
       #Warning.MissingCnd.OP_REST_PareggLong := FALSE;
   END_IF;
   #TON_PareggLong.OP_WORK_MissingCnd.TON(IN := #Ctrl.PareggLong.OP_Work AND NOT #COut.PareggiatoreLong.Work,
                           PT := #Config.DelayMissingCondition);
   IF #TON_PareggLong.OP_WORK_MissingCnd.Q THEN
       #Warning.MissingCnd.OP_WORK_PareggLong := TRUE;   // SR flip-flop
   END_IF;
   IF #Sts.PareggLong.Op_Work_Cnd OR #Ctrl.PareggLong.OP_Rest OR #AreaInterface.RstAlarms THEN
       #Warning.MissingCnd.OP_WORK_PareggLong := FALSE;
   END_IF;
END_REGION

REGION Network 62: [Bloccaggio] - Valve Manager
   RUNG wire#powerrail
      #Bloccaggio(AreaInterface := #AreaInterface, ZSI := #ZSI, DSI := #DSI_OilValve, DataIn :=, Cin :=, Config := #Config.Bloccaggio, Alarm := #Alarm.Bloccaggio, Warning := #Warning.Bloccaggio, MachineInterface =>, COut => #COut.Bloccaggio, DataOut =>)
   END_RUNG
   // the same network as SCL:
   #Bloccaggio(AreaInterface := #AreaInterface,   // "ValveMachine_FB"
               ZSI := #ZSI,
               DSI := #DSI_OilValve,
               Config := #Config.Bloccaggio,
               Alarm := #Alarm.Bloccaggio,
               Warning := #Warning.Bloccaggio,
               COut => #COut.Bloccaggio);
END_REGION

REGION Network 63: [Battuta Vrt ] - Valve Manager
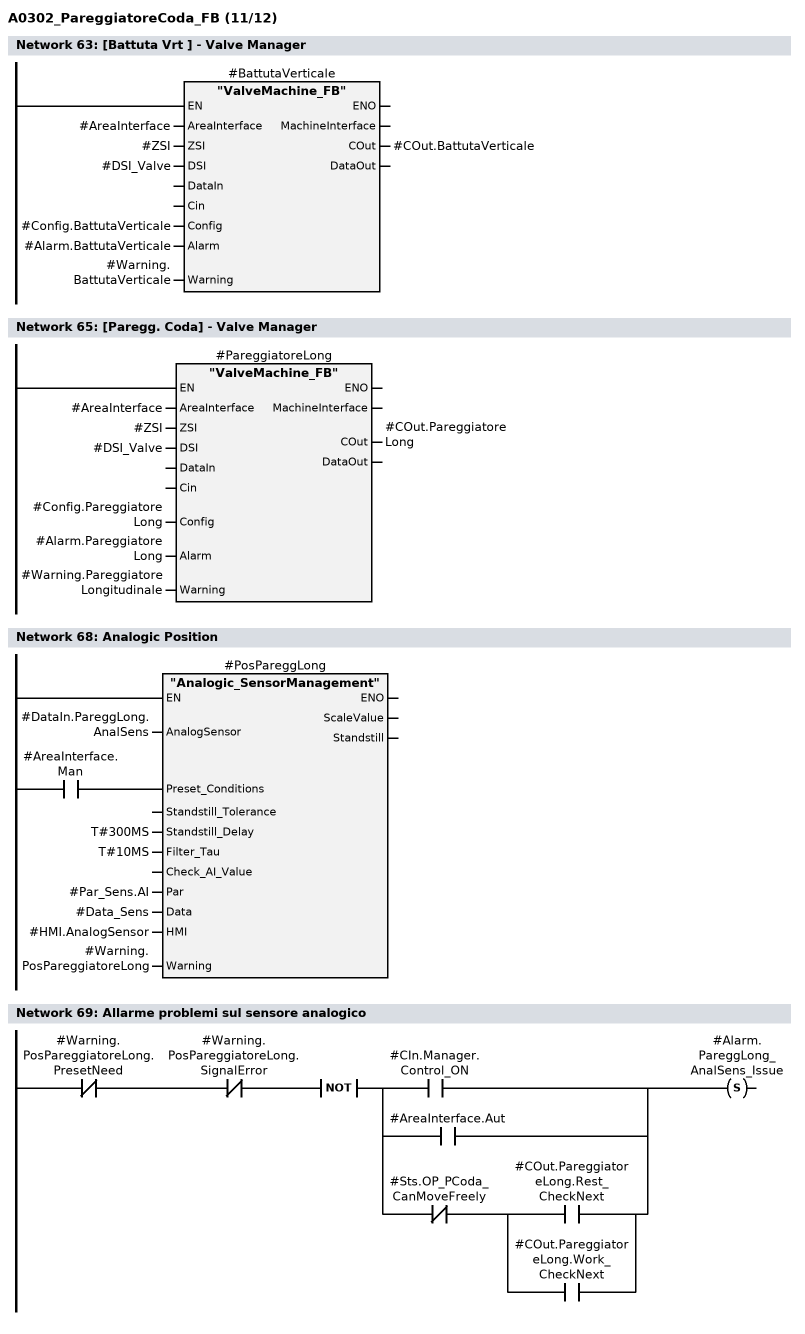
   RUNG wire#powerrail
      #BattutaVerticale(AreaInterface := #AreaInterface, ZSI := #ZSI, DSI := #DSI_Valve, DataIn :=, Cin :=, Config := #Config.BattutaVerticale, Alarm := #Alarm.BattutaVerticale, Warning := #Warning.BattutaVerticale, MachineInterface =>, COut => #COut.BattutaVerticale, DataOut =>)
   END_RUNG
   // the same network as SCL:
   #BattutaVerticale(AreaInterface := #AreaInterface,   // "ValveMachine_FB"
                     ZSI := #ZSI,
                     DSI := #DSI_Valve,
                     Config := #Config.BattutaVerticale,
                     Alarm := #Alarm.BattutaVerticale,
                     Warning := #Warning.BattutaVerticale,
                     COut => #COut.BattutaVerticale);
END_REGION

REGION Network 64 (SCL): [Battuta Vrt ] - Anticipo COut
   #COut.BattutaVerticale := #BattutaVerticale.COut;

   #COut.BattutaVerticale.Rest := #BattutaVerticale.COut.Rest OR #TON_Anticipi.Rest.BattutaVrt.Q;
   #COut.BattutaVerticale.Work := #BattutaVerticale.COut.Work OR #TON_Anticipi.Work.BattutaVrt.Q;
END_REGION

REGION Network 65: [Paregg. Coda] - Valve Manager
   RUNG wire#powerrail
      #PareggiatoreLong(AreaInterface := #AreaInterface, ZSI := #ZSI, DSI := #DSI_Valve, DataIn :=, Cin :=, Config := #Config.PareggiatoreLong, Alarm := #Alarm.PareggiatoreLong, Warning := #Warning.PareggiatoreLongitudinale, MachineInterface =>, COut => #COut.PareggiatoreLong, DataOut =>)
   END_RUNG
   // the same network as SCL:
   #PareggiatoreLong(AreaInterface := #AreaInterface,   // "ValveMachine_FB"
                     ZSI := #ZSI,
                     DSI := #DSI_Valve,
                     Config := #Config.PareggiatoreLong,
                     Alarm := #Alarm.PareggiatoreLong,
                     Warning := #Warning.PareggiatoreLongitudinale,
                     COut => #COut.PareggiatoreLong);
END_REGION

REGION Network 66 (SCL): [Paregg. Coda] - Anticipo COut
   #COut.PareggiatoreLong := #PareggiatoreLong.COut;

   #COut.PareggiatoreLong.Rest := #PareggiatoreLong.COut.Rest OR #TON_Anticipi.Rest.PareggLong.Q;
   #COut.PareggiatoreLong.Work := #PareggiatoreLong.COut.Work OR #TON_Anticipi.Work.PareggLong.Q;
END_REGION

REGION Network 68: Analogic Position
   RUNG wire#powerrail
      #PosPareggLong(Preset_Conditions := wire#w1, AnalogSensor := #DataIn.PareggLong.AnalSens, Standstill_Tolerance :=, Standstill_Delay := T#300MS, Filter_Tau := T#10MS, Check_AI_Value :=, Par := #Par_Sens.AI, Data := #Data_Sens, HMI := #HMI.AnalogSensor, Warning := #Warning.PosPareggiatoreLong, ScaleValue =>, Standstill =>)
   END_RUNG
   RUNG wire#powerrail
      Contact( #AreaInterface.Man )
   END_RUNG wire#w1
   // the same network as SCL:
   #PosPareggLong(AnalogSensor := #DataIn.PareggLong.AnalSens,   // "Analogic_SensorManagement"
                  Preset_Conditions := #AreaInterface.Man,
                  Standstill_Delay := T#300MS,
                  Filter_Tau := T#10MS,
                  Par := #Par_Sens.AI,
                  Data := #Data_Sens,
                  HMI := #HMI.AnalogSensor,
                  Warning := #Warning.PosPareggiatoreLong);
END_REGION

REGION Network 69: Allarme problemi sul sensore analogico
   RUNG wire#powerrail
      I_Contact( #Warning.PosPareggiatoreLong.PresetNeed )
      I_Contact( #Warning.PosPareggiatoreLong.SignalError )
      Not()
      wire#w1
      Contact( #CIn.Manager.Control_ON )
      wire#w2
      S_Coil( #Alarm.PareggLong_AnalSens_Issue )
   END_RUNG
   RUNG wire#w1
      Contact( #AreaInterface.Aut )
   END_RUNG wire#w2
   RUNG wire#w1
      I_Contact( #Sts.OP_PCoda_CanMoveFreely )
      wire#w3
      Contact( #COut.PareggiatoreLong.Rest_CheckNext )
   END_RUNG wire#w2
   RUNG wire#w3
      Contact( #COut.PareggiatoreLong.Work_CheckNext )
   END_RUNG wire#w2
   // the same network as SCL:
   IF NOT (NOT #Warning.PosPareggiatoreLong.PresetNeed AND NOT #Warning.PosPareggiatoreLong.SignalError) AND (#CIn.Manager.Control_ON OR #AreaInterface.Aut OR (NOT #Sts.OP_PCoda_CanMoveFreely AND (#COut.PareggiatoreLong.Rest_CheckNext OR #COut.PareggiatoreLong.Work_CheckNext))) THEN
       #Alarm.PareggLong_AnalSens_Issue := TRUE;
   END_IF;
END_REGION

REGION Network 70 (SCL): PAREGGIAMENTO - Controllo che il Pareggiatore è a lavoro
       // *****************************************************************************************************************************
       // Calcolo lo spazio di sicurezza se ho eseguito il preset del sensore
       // Spazio di frenata da raggiungere

       #Par_Sens.AI.Enable := TRUE;

       IF #Par_Sens.AI.Enable AND #Data_Sens.OffsetValid THEN
           IF #CIn.CarroPareggCoda.Pareggia AND
               #PareggiatoreLong.Cin.Manager.Work AND
               NOT #PareggiatoreLong.DataIn.Rest_Ls[1] AND #PosPareggLong.Standstill
               AND (#PosPareggLong.ScaleValue > #Config.PosPareggiatore.QuotaMin_Work) AND (#PosPareggLong.ScaleValue < #Config.PosPareggiatore.QuotaMax_Work) THEN
               #Ctrl.PareggLong.CheckMesure := TRUE;
           END_IF;

           IF (#PareggiatoreLong.Cin.Manager.Rest OR #PareggiatoreLong.DataIn.Rest_Ls[1])THEN
               #Ctrl.PareggLong.CheckMesure := FALSE;
           END_IF;
       ELSE
           #Ctrl.PareggLong.CheckMesure := FALSE;
       END_IF;
END_REGION

REGION Network 72: <<< MACHINE STATUS >>>
END_REGION

REGION Network 73: Collect machine to zone interface (internal machines OR)
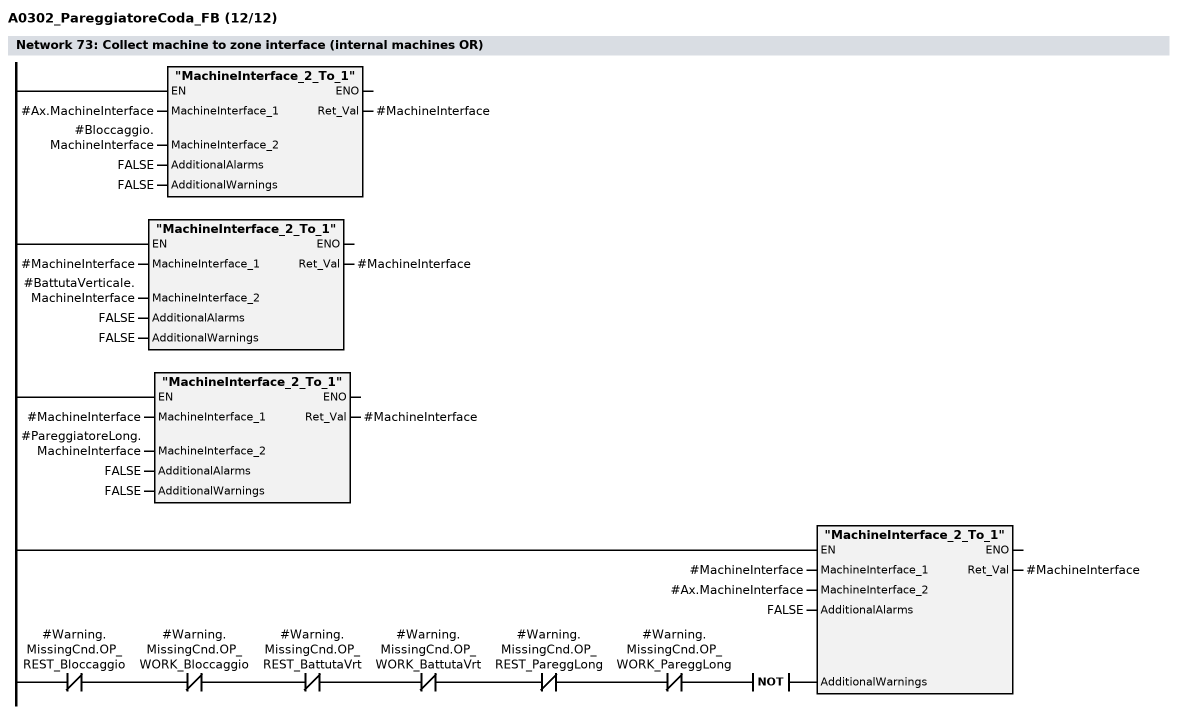
   RUNG wire#powerrail
      "MachineInterface_2_To_1"(MachineInterface_1 := #Ax.MachineInterface, MachineInterface_2 := #Bloccaggio.MachineInterface, AdditionalAlarms := FALSE, AdditionalWarnings := FALSE, Ret_Val => #MachineInterface)
   END_RUNG
   RUNG wire#powerrail
      "MachineInterface_2_To_1"(MachineInterface_1 := #MachineInterface, MachineInterface_2 := #BattutaVerticale.MachineInterface, AdditionalAlarms := FALSE, AdditionalWarnings := FALSE, Ret_Val => #MachineInterface)
   END_RUNG
   RUNG wire#powerrail
      "MachineInterface_2_To_1"(MachineInterface_1 := #MachineInterface, MachineInterface_2 := #PareggiatoreLong.MachineInterface, AdditionalAlarms := FALSE, AdditionalWarnings := FALSE, Ret_Val => #MachineInterface)
   END_RUNG
   RUNG wire#powerrail
      "MachineInterface_2_To_1"(AdditionalWarnings := wire#w1, MachineInterface_1 := #MachineInterface, MachineInterface_2 := #Ax.MachineInterface, AdditionalAlarms := FALSE, Ret_Val => #MachineInterface)
   END_RUNG
   RUNG wire#powerrail
      I_Contact( #Warning.MissingCnd.OP_REST_Bloccaggio )
      I_Contact( #Warning.MissingCnd.OP_WORK_Bloccaggio )
      I_Contact( #Warning.MissingCnd.OP_REST_BattutaVrt )
      I_Contact( #Warning.MissingCnd.OP_WORK_BattutaVrt )
      I_Contact( #Warning.MissingCnd.OP_REST_PareggLong )
      I_Contact( #Warning.MissingCnd.OP_WORK_PareggLong )
      Not()
   END_RUNG wire#w1
   // the same network as SCL:
   #MachineInterface := "MachineInterface_2_To_1"(MachineInterface_1 := #Ax.MachineInterface,
                           MachineInterface_2 := #Bloccaggio.MachineInterface,
                           AdditionalAlarms := FALSE,
                           AdditionalWarnings := FALSE);
   #MachineInterface := "MachineInterface_2_To_1"(MachineInterface_1 := #MachineInterface,
                           MachineInterface_2 := #BattutaVerticale.MachineInterface,
                           AdditionalAlarms := FALSE,
                           AdditionalWarnings := FALSE);
   #MachineInterface := "MachineInterface_2_To_1"(MachineInterface_1 := #MachineInterface,
                           MachineInterface_2 := #PareggiatoreLong.MachineInterface,
                           AdditionalAlarms := FALSE,
                           AdditionalWarnings := FALSE);
   #MachineInterface := "MachineInterface_2_To_1"(MachineInterface_1 := #MachineInterface,
                           MachineInterface_2 := #Ax.MachineInterface,
                           AdditionalAlarms := FALSE,
                           AdditionalWarnings := NOT (NOT #Warning.MissingCnd.OP_REST_Bloccaggio AND NOT #Warning.MissingCnd.OP_WORK_Bloccaggio AND NOT #Warning.MissingCnd.OP_REST_BattutaVrt AND NOT #Warning.MissingCnd.OP_WORK_BattutaVrt AND NOT #Warning.MissingCnd.OP_REST_PareggLong AND NOT #Warning.MissingCnd.OP_WORK_PareggLong));
END_REGION
END_FUNCTION_BLOCK
